Staubli VAL3: Carre10.dtx

public frame fReference = {x=1508.007, y=227.412, z=-659.53, rz=90, fatherId=world[0]}
public jointRx jPark = {j3=90, j5=90}
public jointRx jJoint = {j1=0.56611, j2=53.82368, j3=72.5366, j5=53.63971, j6=175.60048}
public mdesc mNomSpeed = {blend=off}
public mdesc mSpeed[30]
  [0] = {tmax=30, rmax=100, leave=0.1, reach=0.1, blend=cartesian}
  [1] = {tmax=30, rmax=100, leave=0.1, reach=0.1, blend=cartesian}
  [2] = {tmax=30, rmax=100, leave=0.1, reach=0.1, blend=cartesian}
  [3] = {tmax=30, rmax=100, leave=0.1, reach=0.1, blend=cartesian}
  [4] = {tmax=30, rmax=100, leave=0.1, reach=0.1, blend=cartesian}
  [5] = {tmax=30, rmax=100, leave=0.1, reach=0.1, blend=cartesian}
  [6] = {tmax=30, rmax=100, leave=0.1, reach=0.1, blend=cartesian}
  [7] = {tmax=30, rmax=100, leave=0.1, reach=0.1, blend=cartesian}
  [8] = {tmax=30, rmax=100, leave=0.1, reach=0.1, blend=cartesian}
  [9] = {tmax=30, rmax=100, leave=0.1, reach=0.1, blend=cartesian}
  [10] = {tmax=30, rmax=100, leave=0.1, reach=0.1, blend=cartesian}
  [11] = {tmax=30, rmax=100, leave=0.1, reach=0.1, blend=cartesian}
  [12] = {tmax=30, rmax=100, leave=0.1, reach=0.1, blend=cartesian}
  [13] = {tmax=30, rmax=100, leave=0.1, reach=0.1, blend=cartesian}
  [14] = {tmax=30, rmax=100, leave=0.1, reach=0.1, blend=cartesian}
  [15] = {tmax=30, rmax=100, leave=0.1, reach=0.1, blend=cartesian}
  [16] = {tmax=30, rmax=100, leave=0.1, reach=0.1, blend=cartesian}
  [17] = {tmax=30, rmax=100, leave=0.1, reach=0.1, blend=cartesian}
  [18] = {tmax=30, rmax=100, leave=0.1, reach=0.1, blend=cartesian}
  [19] = {tmax=30, rmax=100, leave=0.1, reach=0.1, blend=cartesian}
  [20] = {tmax=30, rmax=100, leave=0.1, reach=0.1, blend=cartesian}
  [21] = {tmax=30, rmax=100, leave=0.1, reach=0.1, blend=cartesian}
  [22] = {tmax=30, rmax=100, leave=0.1, reach=0.1, blend=cartesian}
  [23] = {tmax=30, rmax=100, leave=0.1, reach=0.1, blend=cartesian}
  [24] = {tmax=30, rmax=100, leave=0.1, reach=0.1, blend=cartesian}
  [25] = {tmax=30, rmax=100, leave=0.1, reach=0.1, blend=cartesian}
  [26] = {tmax=30, rmax=100, leave=0.1, reach=0.1, blend=cartesian}
  [27] = {tmax=30, rmax=100, leave=0.1, reach=0.1, blend=cartesian}
  [28] = {tmax=30, rmax=100, leave=0.1, reach=0.1, blend=cartesian}
  [29] = {tmax=30, rmax=100, leave=0.1, reach=0.1, blend=cartesian}
public num nTraj
num nTimeStop
num nTimeStart
num nMode
num nEtat
public pointRx pPoint[1630]
  [0] = {x=-211, y=-153, z=100, rx=-180, rz=85.034, shoulder=lefty, elbow=epositive, wrist=wpositive, fatherId=fReference[0]}
  [1] = {x=-211, y=-153, rx=-180, rz=85.034, shoulder=lefty, elbow=epositive, wrist=wpositive, fatherId=fReference[0]}
  [2] = {x=-211, y=-153, rx=-180, rz=85.034, shoulder=lefty, elbow=epositive, wrist=wpositive, fatherId=fReference[0]}
  [3] = {x=-210.131, y=-163.003, rx=-180, rz=75.103, shoulder=lefty, elbow=epositive, wrist=wpositive, fatherId=fReference[0]}
  [4] = {x=-207.55, y=-172.706, rx=-180, rz=65.172, shoulder=lefty, elbow=epositive, wrist=wpositive, fatherId=fReference[0]}
  [5] = {x=-203.334, y=-181.819, rx=-180, rz=55.241, shoulder=lefty, elbow=epositive, wrist=wpositive, fatherId=fReference[0]}
  [6] = {x=-197.609, y=-190.068, rx=-180, rz=45.309, shoulder=lefty, elbow=epositive, wrist=wpositive, fatherId=fReference[0]}
  [7] = {x=-190.548, y=-197.206, rx=-180, rz=35.378, shoulder=lefty, elbow=epositive, wrist=wpositive, fatherId=fReference[0]}
  [8] = {x=-182.361, y=-203.019, rx=-180, rz=25.447, shoulder=lefty, elbow=epositive, wrist=wpositive, fatherId=fReference[0]}
  [9] = {x=-173.294, y=-207.334, rx=180, rz=15.516, shoulder=lefty, elbow=epositive, wrist=wpositive, fatherId=fReference[0]}
  [10] = {x=-163.619, y=-210.02, rx=-180, rz=5.584, shoulder=lefty, elbow=epositive, wrist=wpositive, fatherId=fReference[0]}
  [11] = {x=-153.626, y=-210.997, rx=-180, rz=0.019, shoulder=lefty, elbow=epositive, wrist=wpositive, fatherId=fReference[0]}
  [12] = {x=-143.573, y=-211, rx=180, shoulder=lefty, elbow=epositive, wrist=wpositive, fatherId=fReference[0]}
  [13] = {x=-133.52, y=-211, rx=180, shoulder=lefty, elbow=epositive, wrist=wpositive, fatherId=fReference[0]}
  [14] = {x=-123.466, y=-211, rx=180, shoulder=lefty, elbow=epositive, wrist=wpositive, fatherId=fReference[0]}
  [15] = {x=-113.413, y=-211, rx=-180, shoulder=lefty, elbow=epositive, wrist=wpositive, fatherId=fReference[0]}
  [16] = {x=-103.36, y=-211, rx=180, shoulder=lefty, elbow=epositive, wrist=wpositive, fatherId=fReference[0]}
  [17] = {x=-93.306, y=-211, rx=-180, shoulder=lefty, elbow=epositive, wrist=wpositive, fatherId=fReference[0]}
  [18] = {x=-83.253, y=-211, rx=-180, shoulder=lefty, elbow=epositive, wrist=wpositive, fatherId=fReference[0]}
  [19] = {x=-73.2, y=-211, rx=-180, shoulder=lefty, elbow=epositive, wrist=wpositive, fatherId=fReference[0]}
  [20] = {x=-63.146, y=-211, rx=180, shoulder=lefty, elbow=epositive, wrist=wpositive, fatherId=fReference[0]}
  [21] = {x=-53.093, y=-211, rx=-180, shoulder=lefty, elbow=epositive, wrist=wpositive, fatherId=fReference[0]}
  [22] = {x=-43.04, y=-211, rx=180, shoulder=lefty, elbow=epositive, wrist=wpositive, fatherId=fReference[0]}
  [23] = {x=-32.986, y=-211, rx=180, shoulder=lefty, elbow=epositive, wrist=wpositive, fatherId=fReference[0]}
  [24] = {x=-22.933, y=-211, rx=-180, shoulder=lefty, elbow=epositive, wrist=wpositive, fatherId=fReference[0]}
  [25] = {x=-12.88, y=-211, rx=-180, shoulder=lefty, elbow=epositive, wrist=wpositive, fatherId=fReference[0]}
  [26] = {x=-2.826, y=-211, rx=180, shoulder=lefty, elbow=epositive, wrist=wpositive, fatherId=fReference[0]}
  [27] = {x=7.227, y=-211, rx=-180, shoulder=lefty, elbow=epositive, wrist=wpositive, fatherId=fReference[0]}
  [28] = {x=17.28, y=-211, rx=-180, shoulder=lefty, elbow=epositive, wrist=wpositive, fatherId=fReference[0]}
  [29] = {x=27.333, y=-211, rx=-180, shoulder=lefty, elbow=epositive, wrist=wpositive, fatherId=fReference[0]}
  [30] = {x=37.387, y=-211, rx=180, shoulder=lefty, elbow=epositive, wrist=wpositive, fatherId=fReference[0]}
  [31] = {x=47.44, y=-211, rx=-180, shoulder=lefty, elbow=epositive, wrist=wpositive, fatherId=fReference[0]}
  [32] = {x=57.493, y=-211, rx=180, shoulder=lefty, elbow=epositive, wrist=wpositive, fatherId=fReference[0]}
  [33] = {x=67.547, y=-211, rx=-180, shoulder=lefty, elbow=epositive, wrist=wpositive, fatherId=fReference[0]}
  [34] = {x=77.6, y=-211, rx=180, shoulder=lefty, elbow=epositive, wrist=wpositive, fatherId=fReference[0]}
  [35] = {x=87.653, y=-211, rx=-180, shoulder=lefty, elbow=epositive, wrist=wpositive, fatherId=fReference[0]}
  [36] = {x=97.707, y=-211, rx=-180, shoulder=lefty, elbow=epositive, wrist=wpositive, fatherId=fReference[0]}
  [37] = {x=107.76, y=-211, rx=180, shoulder=lefty, elbow=epositive, wrist=wpositive, fatherId=fReference[0]}
  [38] = {x=117.813, y=-211, rx=180, shoulder=lefty, elbow=epositive, wrist=wpositive, fatherId=fReference[0]}
  [39] = {x=127.867, y=-211, rx=-180, shoulder=lefty, elbow=epositive, wrist=wpositive, fatherId=fReference[0]}
  [40] = {x=137.92, y=-211, rx=-180, shoulder=lefty, elbow=epositive, wrist=wpositive, fatherId=fReference[0]}
  [41] = {x=147.973, y=-211, rx=-180, rz=-1.241, shoulder=lefty, elbow=epositive, wrist=wpositive, fatherId=fReference[0]}
  [42] = {x=158.02, y=-210.782, rx=-180, rz=-9.931, shoulder=lefty, elbow=epositive, wrist=wpositive, fatherId=fReference[0]}
  [43] = {x=167.911, y=-209.051, rx=-180, rz=-19.863, shoulder=lefty, elbow=epositive, wrist=wpositive, fatherId=fReference[0]}
  [44] = {x=177.354, y=-205.639, rx=-180, rz=-29.794, shoulder=lefty, elbow=epositive, wrist=wpositive, fatherId=fReference[0]}
  [45] = {x=186.068, y=-200.65, rx=180, rz=-39.725, shoulder=lefty, elbow=epositive, wrist=wpositive, fatherId=fReference[0]}
  [46] = {x=193.79, y=-194.233, rx=180, rz=-49.656, shoulder=lefty, elbow=epositive, wrist=wpositive, fatherId=fReference[0]}
  [47] = {x=200.29, y=-186.58, rx=180, rz=-59.588, shoulder=lefty, elbow=epositive, wrist=wpositive, fatherId=fReference[0]}
  [48] = {x=205.373, y=-177.921, rx=180, rz=-69.519, shoulder=lefty, elbow=epositive, wrist=wpositive, fatherId=fReference[0]}
  [49] = {x=208.886, y=-168.515, rx=180, rz=-79.45, shoulder=lefty, elbow=epositive, wrist=wpositive, fatherId=fReference[0]}
  [50] = {x=210.725, y=-158.644, rx=180, rz=-88.43, shoulder=lefty, elbow=epositive, wrist=wpositive, fatherId=fReference[0]}
  [51] = {x=211, y=-148.6, rx=180, rz=-90, shoulder=lefty, elbow=epositive, wrist=wpositive, fatherId=fReference[0]}
  [52] = {x=211, y=-138.546, rx=180, rz=-90, shoulder=lefty, elbow=epositive, wrist=wpositive, fatherId=fReference[0]}
  [53] = {x=211, y=-128.493, rx=180, rz=-90, shoulder=lefty, elbow=epositive, wrist=wpositive, fatherId=fReference[0]}
  [54] = {x=211, y=-118.44, rx=180, rz=-90, shoulder=lefty, elbow=epositive, wrist=wpositive, fatherId=fReference[0]}
  [55] = {x=211, y=-108.386, rx=180, rz=-90, shoulder=lefty, elbow=epositive, wrist=wpositive, fatherId=fReference[0]}
  [56] = {x=211, y=-98.333, rx=180, rz=-90, shoulder=lefty, elbow=epositive, wrist=wpositive, fatherId=fReference[0]}
  [57] = {x=211, y=-88.28, rx=180, rz=-90, shoulder=lefty, elbow=epositive, wrist=wpositive, fatherId=fReference[0]}
  [58] = {x=211, y=-78.226, rx=180, rz=-90, shoulder=lefty, elbow=epositive, wrist=wpositive, fatherId=fReference[0]}
  [59] = {x=211, y=-68.173, rx=180, rz=-90, shoulder=lefty, elbow=epositive, wrist=wpositive, fatherId=fReference[0]}
  [60] = {x=211, y=-58.12, rx=180, rz=-90, shoulder=lefty, elbow=epositive, wrist=wpositive, fatherId=fReference[0]}
  [61] = {x=211, y=-48.066, rx=180, rz=-90, shoulder=lefty, elbow=epositive, wrist=wpositive, fatherId=fReference[0]}
  [62] = {x=211, y=-38.013, rx=180, rz=-90, shoulder=lefty, elbow=epositive, wrist=wpositive, fatherId=fReference[0]}
  [63] = {x=211, y=-27.96, rx=180, rz=-90, shoulder=lefty, elbow=epositive, wrist=wpositive, fatherId=fReference[0]}
  [64] = {x=211, y=-17.906, rx=180, rz=-90, shoulder=lefty, elbow=epositive, wrist=wpositive, fatherId=fReference[0]}
  [65] = {x=211, y=-7.853, rx=180, rz=-90, shoulder=lefty, elbow=epositive, wrist=wpositive, fatherId=fReference[0]}
  [66] = {x=211, y=2.2, rx=180, rz=-90, shoulder=lefty, elbow=epositive, wrist=wpositive, fatherId=fReference[0]}
  [67] = {x=211, y=12.254, rx=180, rz=-90, shoulder=lefty, elbow=epositive, wrist=wpositive, fatherId=fReference[0]}
  [68] = {x=211, y=22.307, rx=180, rz=-90, shoulder=lefty, elbow=epositive, wrist=wpositive, fatherId=fReference[0]}
  [69] = {x=211, y=32.36, rx=180, rz=-90, shoulder=lefty, elbow=epositive, wrist=wpositive, fatherId=fReference[0]}
  [70] = {x=211, y=42.413, rx=180, rz=-90, shoulder=lefty, elbow=epositive, wrist=wpositive, fatherId=fReference[0]}
  [71] = {x=211, y=52.467, rx=180, rz=-90, shoulder=lefty, elbow=epositive, wrist=wpositive, fatherId=fReference[0]}
  [72] = {x=211, y=62.52, rx=180, rz=-90, shoulder=lefty, elbow=epositive, wrist=wpositive, fatherId=fReference[0]}
  [73] = {x=211, y=72.573, rx=180, rz=-90, shoulder=lefty, elbow=epositive, wrist=wpositive, fatherId=fReference[0]}
  [74] = {x=211, y=82.627, rx=180, rz=-90, shoulder=lefty, elbow=epositive, wrist=wpositive, fatherId=fReference[0]}
  [75] = {x=211, y=92.68, rx=180, rz=-90, shoulder=lefty, elbow=epositive, wrist=wpositive, fatherId=fReference[0]}
  [76] = {x=211, y=102.733, rx=180, rz=-90, shoulder=lefty, elbow=epositive, wrist=wpositive, fatherId=fReference[0]}
  [77] = {x=211, y=112.787, rx=180, rz=-90, shoulder=lefty, elbow=epositive, wrist=wpositive, fatherId=fReference[0]}
  [78] = {x=211, y=122.84, rx=180, rz=-90, shoulder=lefty, elbow=epositive, wrist=wpositive, fatherId=fReference[0]}
  [79] = {x=211, y=132.893, rx=180, rz=-90, shoulder=lefty, elbow=epositive, wrist=wpositive, fatherId=fReference[0]}
  [80] = {x=211, y=142.947, rx=180, rz=-90, shoulder=lefty, elbow=epositive, wrist=wpositive, fatherId=fReference[0]}
  [81] = {x=211, y=153, rx=-180, rz=-94.966, shoulder=lefty, elbow=epositive, wrist=wpositive, fatherId=fReference[0]}
  [82] = {x=210.131, y=163.003, rx=-180, rz=-104.897, shoulder=lefty, elbow=epositive, wrist=wpositive, fatherId=fReference[0]}
  [83] = {x=207.55, y=172.706, rx=-180, rz=-114.828, shoulder=lefty, elbow=epositive, wrist=wpositive, fatherId=fReference[0]}
  [84] = {x=203.334, y=181.819, rx=-180, rz=-124.759, shoulder=lefty, elbow=epositive, wrist=wpositive, fatherId=fReference[0]}
  [85] = {x=197.609, y=190.068, rx=-180, rz=-134.691, shoulder=lefty, elbow=epositive, wrist=wpositive, fatherId=fReference[0]}
  [86] = {x=190.548, y=197.206, rx=180, rz=-144.622, shoulder=lefty, elbow=epositive, wrist=wpositive, fatherId=fReference[0]}
  [87] = {x=182.361, y=203.019, rx=-180, rz=-154.553, shoulder=lefty, elbow=epositive, wrist=wpositive, fatherId=fReference[0]}
  [88] = {x=173.294, y=207.334, rx=-180, rz=-164.484, shoulder=lefty, elbow=epositive, wrist=wpositive, fatherId=fReference[0]}
  [89] = {x=163.619, y=210.02, rx=-180, rz=-174.416, shoulder=lefty, elbow=epositive, wrist=wpositive, fatherId=fReference[0]}
  [90] = {x=153.626, y=210.997, rx=-180, rz=-179.981, shoulder=lefty, elbow=epositive, wrist=wpositive, fatherId=fReference[0]}
  [91] = {x=143.573, y=211, rx=180, rz=-180, shoulder=lefty, elbow=epositive, wrist=wpositive, fatherId=fReference[0]}
  [92] = {x=133.52, y=211, rx=-180, rz=180, shoulder=lefty, elbow=epositive, wrist=wpositive, fatherId=fReference[0]}
  [93] = {x=123.466, y=211, rx=-180, rz=180, shoulder=lefty, elbow=epositive, wrist=wpositive, fatherId=fReference[0]}
  [94] = {x=113.413, y=211, rx=180, rz=-180, shoulder=lefty, elbow=epositive, wrist=wpositive, fatherId=fReference[0]}
  [95] = {x=103.36, y=211, rx=180, rz=180, shoulder=lefty, elbow=epositive, wrist=wpositive, fatherId=fReference[0]}
  [96] = {x=93.306, y=211, rx=-180, rz=180, shoulder=lefty, elbow=epositive, wrist=wpositive, fatherId=fReference[0]}
  [97] = {x=83.253, y=211, rx=-180, rz=-180, shoulder=lefty, elbow=epositive, wrist=wpositive, fatherId=fReference[0]}
  [98] = {x=73.2, y=211, rx=180, rz=180, shoulder=lefty, elbow=epositive, wrist=wpositive, fatherId=fReference[0]}
  [99] = {x=63.146, y=211, rx=-180, rz=180, shoulder=lefty, elbow=epositive, wrist=wpositive, fatherId=fReference[0]}
  [100] = {x=53.093, y=211, rx=-180, rz=180, shoulder=lefty, elbow=epositive, wrist=wpositive, fatherId=fReference[0]}
  [101] = {x=43.04, y=211, rx=-180, rz=180, shoulder=lefty, elbow=epositive, wrist=wpositive, fatherId=fReference[0]}
  [102] = {x=32.986, y=211, rx=-180, rz=180, shoulder=lefty, elbow=epositive, wrist=wpositive, fatherId=fReference[0]}
  [103] = {x=22.933, y=211, rx=-180, rz=180, shoulder=lefty, elbow=epositive, wrist=wpositive, fatherId=fReference[0]}
  [104] = {x=12.88, y=211, rx=180, rz=180, shoulder=lefty, elbow=epositive, wrist=wpositive, fatherId=fReference[0]}
  [105] = {x=2.826, y=211, rx=180, rz=180, shoulder=lefty, elbow=epositive, wrist=wpositive, fatherId=fReference[0]}
  [106] = {x=-7.227, y=211, rx=-180, rz=180, shoulder=lefty, elbow=epositive, wrist=wpositive, fatherId=fReference[0]}
  [107] = {x=-17.28, y=211, rx=180, rz=180, shoulder=lefty, elbow=epositive, wrist=wpositive, fatherId=fReference[0]}
  [108] = {x=-27.333, y=211, rx=180, rz=180, shoulder=lefty, elbow=epositive, wrist=wpositive, fatherId=fReference[0]}
  [109] = {x=-37.387, y=211, rx=-180, rz=180, shoulder=lefty, elbow=epositive, wrist=wpositive, fatherId=fReference[0]}
  [110] = {x=-47.44, y=211, rx=180, rz=180, shoulder=lefty, elbow=epositive, wrist=wpositive, fatherId=fReference[0]}
  [111] = {x=-57.493, y=211, rx=-180, rz=180, shoulder=lefty, elbow=epositive, wrist=wpositive, fatherId=fReference[0]}
  [112] = {x=-67.547, y=211, rx=180, rz=180, shoulder=lefty, elbow=epositive, wrist=wpositive, fatherId=fReference[0]}
  [113] = {x=-77.6, y=211, rx=-180, rz=180, shoulder=lefty, elbow=epositive, wrist=wpositive, fatherId=fReference[0]}
  [114] = {x=-87.653, y=211, rx=180, rz=180, shoulder=lefty, elbow=epositive, wrist=wpositive, fatherId=fReference[0]}
  [115] = {x=-97.707, y=211, rx=180, rz=180, shoulder=lefty, elbow=epositive, wrist=wpositive, fatherId=fReference[0]}
  [116] = {x=-107.76, y=211, rx=180, rz=180, shoulder=lefty, elbow=epositive, wrist=wpositive, fatherId=fReference[0]}
  [117] = {x=-117.813, y=211, rx=-180, rz=180, shoulder=lefty, elbow=epositive, wrist=wpositive, fatherId=fReference[0]}
  [118] = {x=-127.867, y=211, rx=-180, rz=180, shoulder=lefty, elbow=epositive, wrist=wpositive, fatherId=fReference[0]}
  [119] = {x=-137.92, y=211, rx=180, rz=180, shoulder=lefty, elbow=epositive, wrist=wpositive, fatherId=fReference[0]}
  [120] = {x=-147.973, y=211, rx=180, rz=178.759, shoulder=lefty, elbow=epositive, wrist=wpositive, fatherId=fReference[0]}
  [121] = {x=-158.02, y=210.782, rx=180, rz=170.069, shoulder=lefty, elbow=epositive, wrist=wpositive, fatherId=fReference[0]}
  [122] = {x=-167.911, y=209.051, rx=180, rz=160.137, shoulder=lefty, elbow=epositive, wrist=wpositive, fatherId=fReference[0]}
  [123] = {x=-177.354, y=205.639, rx=180, rz=150.206, shoulder=lefty, elbow=epositive, wrist=wpositive, fatherId=fReference[0]}
  [124] = {x=-186.068, y=200.65, rx=180, rz=140.275, shoulder=lefty, elbow=epositive, wrist=wpositive, fatherId=fReference[0]}
  [125] = {x=-193.79, y=194.233, rx=-180, rz=130.344, shoulder=lefty, elbow=epositive, wrist=wpositive, fatherId=fReference[0]}
  [126] = {x=-200.29, y=186.58, rx=180, rz=120.412, shoulder=lefty, elbow=epositive, wrist=wpositive, fatherId=fReference[0]}
  [127] = {x=-205.373, y=177.921, rx=180, rz=110.481, shoulder=lefty, elbow=epositive, wrist=wpositive, fatherId=fReference[0]}
  [128] = {x=-208.886, y=168.515, rx=180, rz=100.55, shoulder=lefty, elbow=epositive, wrist=wpositive, fatherId=fReference[0]}
  [129] = {x=-210.725, y=158.644, rx=180, rz=91.57, shoulder=lefty, elbow=epositive, wrist=wpositive, fatherId=fReference[0]}
  [130] = {x=-211, y=148.6, rx=-180, rz=90, shoulder=lefty, elbow=epositive, wrist=wpositive, fatherId=fReference[0]}
  [131] = {x=-211, y=138.546, rx=-180, rz=90, shoulder=lefty, elbow=epositive, wrist=wpositive, fatherId=fReference[0]}
  [132] = {x=-211, y=128.493, rx=-180, rz=90, shoulder=lefty, elbow=epositive, wrist=wpositive, fatherId=fReference[0]}
  [133] = {x=-211, y=118.44, rx=-180, rz=90, shoulder=lefty, elbow=epositive, wrist=wpositive, fatherId=fReference[0]}
  [134] = {x=-211, y=108.386, rx=-180, rz=90, shoulder=lefty, elbow=epositive, wrist=wpositive, fatherId=fReference[0]}
  [135] = {x=-211, y=98.333, rx=-180, rz=90, shoulder=lefty, elbow=epositive, wrist=wpositive, fatherId=fReference[0]}
  [136] = {x=-211, y=88.28, rx=-180, rz=90, shoulder=lefty, elbow=epositive, wrist=wpositive, fatherId=fReference[0]}
  [137] = {x=-211, y=78.226, rx=-180, rz=90, shoulder=lefty, elbow=epositive, wrist=wpositive, fatherId=fReference[0]}
  [138] = {x=-211, y=68.173, rx=-180, rz=90, shoulder=lefty, elbow=epositive, wrist=wpositive, fatherId=fReference[0]}
  [139] = {x=-211, y=58.12, rx=-180, rz=90, shoulder=lefty, elbow=epositive, wrist=wpositive, fatherId=fReference[0]}
  [140] = {x=-211, y=48.066, rx=-180, rz=90, shoulder=lefty, elbow=epositive, wrist=wpositive, fatherId=fReference[0]}
  [141] = {x=-211, y=38.013, rx=-180, rz=90, shoulder=lefty, elbow=epositive, wrist=wpositive, fatherId=fReference[0]}
  [142] = {x=-211, y=27.96, rx=-180, rz=90, shoulder=lefty, elbow=epositive, wrist=wpositive, fatherId=fReference[0]}
  [143] = {x=-211, y=17.906, rx=-180, rz=90, shoulder=lefty, elbow=epositive, wrist=wpositive, fatherId=fReference[0]}
  [144] = {x=-211, y=7.853, rx=-180, rz=90, shoulder=lefty, elbow=epositive, wrist=wpositive, fatherId=fReference[0]}
  [145] = {x=-211, y=-2.2, rx=-180, rz=90, shoulder=lefty, elbow=epositive, wrist=wpositive, fatherId=fReference[0]}
  [146] = {x=-211, y=-12.254, rx=-180, rz=90, shoulder=lefty, elbow=epositive, wrist=wpositive, fatherId=fReference[0]}
  [147] = {x=-211, y=-22.307, rx=-180, rz=90, shoulder=lefty, elbow=epositive, wrist=wpositive, fatherId=fReference[0]}
  [148] = {x=-211, y=-32.36, rx=-180, rz=90, shoulder=lefty, elbow=epositive, wrist=wpositive, fatherId=fReference[0]}
  [149] = {x=-211, y=-42.413, rx=-180, rz=90, shoulder=lefty, elbow=epositive, wrist=wpositive, fatherId=fReference[0]}
  [150] = {x=-211, y=-52.467, rx=-180, rz=90, shoulder=lefty, elbow=epositive, wrist=wpositive, fatherId=fReference[0]}
  [151] = {x=-211, y=-62.52, rx=-180, rz=90, shoulder=lefty, elbow=epositive, wrist=wpositive, fatherId=fReference[0]}
  [152] = {x=-211, y=-72.573, rx=-180, rz=90, shoulder=lefty, elbow=epositive, wrist=wpositive, fatherId=fReference[0]}
  [153] = {x=-211, y=-82.627, rx=-180, rz=90, shoulder=lefty, elbow=epositive, wrist=wpositive, fatherId=fReference[0]}
  [154] = {x=-211, y=-92.68, rx=-180, rz=90, shoulder=lefty, elbow=epositive, wrist=wpositive, fatherId=fReference[0]}
  [155] = {x=-211, y=-102.733, rx=-180, rz=90, shoulder=lefty, elbow=epositive, wrist=wpositive, fatherId=fReference[0]}
  [156] = {x=-211, y=-112.787, rx=-180, rz=90, shoulder=lefty, elbow=epositive, wrist=wpositive, fatherId=fReference[0]}
  [157] = {x=-211, y=-122.84, rx=-180, rz=90, shoulder=lefty, elbow=epositive, wrist=wpositive, fatherId=fReference[0]}
  [158] = {x=-211, y=-132.893, rx=-180, rz=90, shoulder=lefty, elbow=epositive, wrist=wpositive, fatherId=fReference[0]}
  [159] = {x=-211, y=-142.947, rx=-180, rz=90, shoulder=lefty, elbow=epositive, wrist=wpositive, fatherId=fReference[0]}
  [160] = {x=-211, y=-153, rx=-180, rz=90, shoulder=lefty, elbow=epositive, wrist=wpositive, fatherId=fReference[0]}
  [161] = {x=-211, y=-153, rx=-180, rz=90, shoulder=lefty, elbow=epositive, wrist=wpositive, fatherId=fReference[0]}
  [162] = {x=-211, y=-153, z=100, rx=-180, rz=90, shoulder=lefty, elbow=epositive, wrist=wpositive, fatherId=fReference[0]}
  [163] = {x=-211, y=-153, z=122, rx=-180, rz=90, shoulder=lefty, elbow=epositive, wrist=wpositive, fatherId=fReference[0]}
  [164] = {x=-211, y=-153, z=22, rx=-180, rz=90, shoulder=lefty, elbow=epositive, wrist=wpositive, fatherId=fReference[0]}
  [165] = {x=-211, y=-153, z=22, rx=-180, rz=90, shoulder=lefty, elbow=epositive, wrist=wpositive, fatherId=fReference[0]}
  [166] = {x=-211, y=-142.947, z=22, rx=-180, rz=90, shoulder=lefty, elbow=epositive, wrist=wpositive, fatherId=fReference[0]}
  [167] = {x=-211, y=-132.893, z=22, rx=-180, rz=90, shoulder=lefty, elbow=epositive, wrist=wpositive, fatherId=fReference[0]}
  [168] = {x=-211, y=-122.84, z=22, rx=-180, rz=90, shoulder=lefty, elbow=epositive, wrist=wpositive, fatherId=fReference[0]}
  [169] = {x=-211, y=-112.787, z=22, rx=-180, rz=90, shoulder=lefty, elbow=epositive, wrist=wpositive, fatherId=fReference[0]}
  [170] = {x=-211, y=-102.733, z=22, rx=-180, rz=90, shoulder=lefty, elbow=epositive, wrist=wpositive, fatherId=fReference[0]}
  [171] = {x=-211, y=-92.68, z=22, rx=-180, rz=90, shoulder=lefty, elbow=epositive, wrist=wpositive, fatherId=fReference[0]}
  [172] = {x=-211, y=-82.627, z=22, rx=-180, rz=90, shoulder=lefty, elbow=epositive, wrist=wpositive, fatherId=fReference[0]}
  [173] = {x=-211, y=-72.573, z=22, rx=-180, rz=90, shoulder=lefty, elbow=epositive, wrist=wpositive, fatherId=fReference[0]}
  [174] = {x=-211, y=-62.52, z=22, rx=-180, rz=90, shoulder=lefty, elbow=epositive, wrist=wpositive, fatherId=fReference[0]}
  [175] = {x=-211, y=-52.467, z=22, rx=-180, rz=90, shoulder=lefty, elbow=epositive, wrist=wpositive, fatherId=fReference[0]}
  [176] = {x=-211, y=-42.413, z=22, rx=-180, rz=90, shoulder=lefty, elbow=epositive, wrist=wpositive, fatherId=fReference[0]}
  [177] = {x=-211, y=-32.36, z=22, rx=-180, rz=90, shoulder=lefty, elbow=epositive, wrist=wpositive, fatherId=fReference[0]}
  [178] = {x=-211, y=-22.307, z=22, rx=-180, rz=90, shoulder=lefty, elbow=epositive, wrist=wpositive, fatherId=fReference[0]}
  [179] = {x=-211, y=-12.254, z=22, rx=-180, rz=90, shoulder=lefty, elbow=epositive, wrist=wpositive, fatherId=fReference[0]}
  [180] = {x=-211, y=-2.2, z=22, rx=-180, rz=90, shoulder=lefty, elbow=epositive, wrist=wpositive, fatherId=fReference[0]}
  [181] = {x=-211, y=7.853, z=22, rx=-180, rz=90, shoulder=lefty, elbow=epositive, wrist=wpositive, fatherId=fReference[0]}
  [182] = {x=-211, y=17.906, z=22, rx=-180, rz=90, shoulder=lefty, elbow=epositive, wrist=wpositive, fatherId=fReference[0]}
  [183] = {x=-211, y=27.96, z=22, rx=-180, rz=90, shoulder=lefty, elbow=epositive, wrist=wpositive, fatherId=fReference[0]}
  [184] = {x=-211, y=38.013, z=22, rx=-180, rz=90, shoulder=lefty, elbow=epositive, wrist=wpositive, fatherId=fReference[0]}
  [185] = {x=-211, y=48.066, z=22, rx=-180, rz=90, shoulder=lefty, elbow=epositive, wrist=wpositive, fatherId=fReference[0]}
  [186] = {x=-211, y=58.12, z=22, rx=-180, rz=90, shoulder=lefty, elbow=epositive, wrist=wpositive, fatherId=fReference[0]}
  [187] = {x=-211, y=68.173, z=22, rx=-180, rz=90, shoulder=lefty, elbow=epositive, wrist=wpositive, fatherId=fReference[0]}
  [188] = {x=-211, y=78.226, z=22, rx=-180, rz=90, shoulder=lefty, elbow=epositive, wrist=wpositive, fatherId=fReference[0]}
  [189] = {x=-211, y=88.28, z=22, rx=-180, rz=90, shoulder=lefty, elbow=epositive, wrist=wpositive, fatherId=fReference[0]}
  [190] = {x=-211, y=98.333, z=22, rx=-180, rz=90, shoulder=lefty, elbow=epositive, wrist=wpositive, fatherId=fReference[0]}
  [191] = {x=-211, y=108.386, z=22, rx=-180, rz=90, shoulder=lefty, elbow=epositive, wrist=wpositive, fatherId=fReference[0]}
  [192] = {x=-211, y=118.44, z=22, rx=-180, rz=90, shoulder=lefty, elbow=epositive, wrist=wpositive, fatherId=fReference[0]}
  [193] = {x=-211, y=128.493, z=22, rx=-180, rz=90, shoulder=lefty, elbow=epositive, wrist=wpositive, fatherId=fReference[0]}
  [194] = {x=-211, y=138.546, z=22, rx=-180, rz=90, shoulder=lefty, elbow=epositive, wrist=wpositive, fatherId=fReference[0]}
  [195] = {x=-211, y=148.6, z=22, rx=180, rz=91.57, shoulder=lefty, elbow=epositive, wrist=wpositive, fatherId=fReference[0]}
  [196] = {x=-210.725, y=158.644, z=22, rx=180, rz=100.55, shoulder=lefty, elbow=epositive, wrist=wpositive, fatherId=fReference[0]}
  [197] = {x=-208.886, y=168.515, z=22, rx=180, rz=110.481, shoulder=lefty, elbow=epositive, wrist=wpositive, fatherId=fReference[0]}
  [198] = {x=-205.373, y=177.921, z=22, rx=180, rz=120.412, shoulder=lefty, elbow=epositive, wrist=wpositive, fatherId=fReference[0]}
  [199] = {x=-200.29, y=186.58, z=22, rx=-180, rz=130.344, shoulder=lefty, elbow=epositive, wrist=wpositive, fatherId=fReference[0]}
  [200] = {x=-193.79, y=194.233, z=22, rx=-180, rz=140.275, shoulder=lefty, elbow=epositive, wrist=wpositive, fatherId=fReference[0]}
  [201] = {x=-186.068, y=200.65, z=22, rx=180, rz=150.206, shoulder=lefty, elbow=epositive, wrist=wpositive, fatherId=fReference[0]}
  [202] = {x=-177.354, y=205.639, z=22, rx=180, rz=160.137, shoulder=lefty, elbow=epositive, wrist=wpositive, fatherId=fReference[0]}
  [203] = {x=-167.911, y=209.051, z=22, rx=180, rz=170.069, shoulder=lefty, elbow=epositive, wrist=wpositive, fatherId=fReference[0]}
  [204] = {x=-158.02, y=210.782, z=22, rx=180, rz=178.759, shoulder=lefty, elbow=epositive, wrist=wpositive, fatherId=fReference[0]}
  [205] = {x=-147.973, y=211, z=22, rx=-180, rz=180, shoulder=lefty, elbow=epositive, wrist=wpositive, fatherId=fReference[0]}
  [206] = {x=-137.92, y=211, z=22, rx=-180, rz=180, shoulder=lefty, elbow=epositive, wrist=wpositive, fatherId=fReference[0]}
  [207] = {x=-127.867, y=211, z=22, rx=-180, rz=180, shoulder=lefty, elbow=epositive, wrist=wpositive, fatherId=fReference[0]}
  [208] = {x=-117.813, y=211, z=22, rx=180, rz=180, shoulder=lefty, elbow=epositive, wrist=wpositive, fatherId=fReference[0]}
  [209] = {x=-107.76, y=211, z=22, rx=180, rz=180, shoulder=lefty, elbow=epositive, wrist=wpositive, fatherId=fReference[0]}
  [210] = {x=-97.707, y=211, z=22, rx=-180, rz=180, shoulder=lefty, elbow=epositive, wrist=wpositive, fatherId=fReference[0]}
  [211] = {x=-87.653, y=211, z=22, rx=-180, rz=180, shoulder=lefty, elbow=epositive, wrist=wpositive, fatherId=fReference[0]}
  [212] = {x=-77.6, y=211, z=22, rx=-180, rz=180, shoulder=lefty, elbow=epositive, wrist=wpositive, fatherId=fReference[0]}
  [213] = {x=-67.547, y=211, z=22, rx=-180, rz=180, shoulder=lefty, elbow=epositive, wrist=wpositive, fatherId=fReference[0]}
  [214] = {x=-57.493, y=211, z=22, rx=180, rz=180, shoulder=lefty, elbow=epositive, wrist=wpositive, fatherId=fReference[0]}
  [215] = {x=-47.44, y=211, z=22, rx=180, rz=180, shoulder=lefty, elbow=epositive, wrist=wpositive, fatherId=fReference[0]}
  [216] = {x=-37.387, y=211, z=22, rx=-180, rz=180, shoulder=lefty, elbow=epositive, wrist=wpositive, fatherId=fReference[0]}
  [217] = {x=-27.333, y=211, z=22, rx=-180, rz=180, shoulder=lefty, elbow=epositive, wrist=wpositive, fatherId=fReference[0]}
  [218] = {x=-17.28, y=211, z=22, rx=180, rz=180, shoulder=lefty, elbow=epositive, wrist=wpositive, fatherId=fReference[0]}
  [219] = {x=-7.227, y=211, z=22, rx=-180, rz=180, shoulder=lefty, elbow=epositive, wrist=wpositive, fatherId=fReference[0]}
  [220] = {x=2.826, y=211, z=22, rx=-180, rz=180, shoulder=lefty, elbow=epositive, wrist=wpositive, fatherId=fReference[0]}
  [221] = {x=12.88, y=211, z=22, rx=-180, rz=180, shoulder=lefty, elbow=epositive, wrist=wpositive, fatherId=fReference[0]}
  [222] = {x=22.933, y=211, z=22, rx=180, rz=180, shoulder=lefty, elbow=epositive, wrist=wpositive, fatherId=fReference[0]}
  [223] = {x=32.986, y=211, z=22, rx=180, rz=180, shoulder=lefty, elbow=epositive, wrist=wpositive, fatherId=fReference[0]}
  [224] = {x=43.04, y=211, z=22, rx=-180, rz=180, shoulder=lefty, elbow=epositive, wrist=wpositive, fatherId=fReference[0]}
  [225] = {x=53.093, y=211, z=22, rx=-180, rz=180, shoulder=lefty, elbow=epositive, wrist=wpositive, fatherId=fReference[0]}
  [226] = {x=63.146, y=211, z=22, rx=-180, rz=180, shoulder=lefty, elbow=epositive, wrist=wpositive, fatherId=fReference[0]}
  [227] = {x=73.2, y=211, z=22, rx=180, rz=180, shoulder=lefty, elbow=epositive, wrist=wpositive, fatherId=fReference[0]}
  [228] = {x=83.253, y=211, z=22, rx=180, rz=-180, shoulder=lefty, elbow=epositive, wrist=wpositive, fatherId=fReference[0]}
  [229] = {x=93.306, y=211, z=22, rx=-180, rz=180, shoulder=lefty, elbow=epositive, wrist=wpositive, fatherId=fReference[0]}
  [230] = {x=103.36, y=211, z=22, rx=180, rz=180, shoulder=lefty, elbow=epositive, wrist=wpositive, fatherId=fReference[0]}
  [231] = {x=113.413, y=211, z=22, rx=180, rz=-180, shoulder=lefty, elbow=epositive, wrist=wpositive, fatherId=fReference[0]}
  [232] = {x=123.466, y=211, z=22, rx=180, rz=180, shoulder=lefty, elbow=epositive, wrist=wpositive, fatherId=fReference[0]}
  [233] = {x=133.52, y=211, z=22, rx=-180, rz=180, shoulder=lefty, elbow=epositive, wrist=wpositive, fatherId=fReference[0]}
  [234] = {x=143.573, y=211, z=22, rx=-180, rz=-179.981, shoulder=lefty, elbow=epositive, wrist=wpositive, fatherId=fReference[0]}
  [235] = {x=153.626, y=210.997, z=22, rx=-180, rz=-174.416, shoulder=lefty, elbow=epositive, wrist=wpositive, fatherId=fReference[0]}
  [236] = {x=163.619, y=210.02, z=22, rx=180, rz=-164.484, shoulder=lefty, elbow=epositive, wrist=wpositive, fatherId=fReference[0]}
  [237] = {x=173.294, y=207.334, z=22, rx=-180, rz=-154.553, shoulder=lefty, elbow=epositive, wrist=wpositive, fatherId=fReference[0]}
  [238] = {x=182.361, y=203.019, z=22, rx=-180, rz=-144.622, shoulder=lefty, elbow=epositive, wrist=wpositive, fatherId=fReference[0]}
  [239] = {x=190.548, y=197.206, z=22, rx=-180, rz=-134.691, shoulder=lefty, elbow=epositive, wrist=wpositive, fatherId=fReference[0]}
  [240] = {x=197.609, y=190.068, z=22, rx=-180, rz=-124.759, shoulder=lefty, elbow=epositive, wrist=wpositive, fatherId=fReference[0]}
  [241] = {x=203.334, y=181.819, z=22, rx=-180, rz=-114.828, shoulder=lefty, elbow=epositive, wrist=wpositive, fatherId=fReference[0]}
  [242] = {x=207.55, y=172.706, z=22, rx=-180, rz=-104.897, shoulder=lefty, elbow=epositive, wrist=wpositive, fatherId=fReference[0]}
  [243] = {x=210.131, y=163.003, z=22, rx=-180, rz=-94.966, shoulder=lefty, elbow=epositive, wrist=wpositive, fatherId=fReference[0]}
  [244] = {x=211, y=153, z=22, rx=180, rz=-90, shoulder=lefty, elbow=epositive, wrist=wpositive, fatherId=fReference[0]}
  [245] = {x=211, y=142.947, z=22, rx=180, rz=-90, shoulder=lefty, elbow=epositive, wrist=wpositive, fatherId=fReference[0]}
  [246] = {x=211, y=132.893, z=22, rx=180, rz=-90, shoulder=lefty, elbow=epositive, wrist=wpositive, fatherId=fReference[0]}
  [247] = {x=211, y=122.84, z=22, rx=-180, rz=-90, shoulder=lefty, elbow=epositive, wrist=wpositive, fatherId=fReference[0]}
  [248] = {x=211, y=112.787, z=22, rx=180, rz=-90, shoulder=lefty, elbow=epositive, wrist=wpositive, fatherId=fReference[0]}
  [249] = {x=211, y=102.733, z=22, rx=180, rz=-90, shoulder=lefty, elbow=epositive, wrist=wpositive, fatherId=fReference[0]}
  [250] = {x=211, y=92.68, z=22, rx=180, rz=-90, shoulder=lefty, elbow=epositive, wrist=wpositive, fatherId=fReference[0]}
  [251] = {x=211, y=82.627, z=22, rx=180, rz=-90, shoulder=lefty, elbow=epositive, wrist=wpositive, fatherId=fReference[0]}
  [252] = {x=211, y=72.573, z=22, rx=180, rz=-90, shoulder=lefty, elbow=epositive, wrist=wpositive, fatherId=fReference[0]}
  [253] = {x=211, y=62.52, z=22, rx=180, rz=-90, shoulder=lefty, elbow=epositive, wrist=wpositive, fatherId=fReference[0]}
  [254] = {x=211, y=52.467, z=22, rx=180, rz=-90, shoulder=lefty, elbow=epositive, wrist=wpositive, fatherId=fReference[0]}
  [255] = {x=211, y=42.413, z=22, rx=180, rz=-90, shoulder=lefty, elbow=epositive, wrist=wpositive, fatherId=fReference[0]}
  [256] = {x=211, y=32.36, z=22, rx=180, rz=-90, shoulder=lefty, elbow=epositive, wrist=wpositive, fatherId=fReference[0]}
  [257] = {x=211, y=22.307, z=22, rx=180, rz=-90, shoulder=lefty, elbow=epositive, wrist=wpositive, fatherId=fReference[0]}
  [258] = {x=211, y=12.254, z=22, rx=180, rz=-90, shoulder=lefty, elbow=epositive, wrist=wpositive, fatherId=fReference[0]}
  [259] = {x=211, y=2.2, z=22, rx=180, rz=-90, shoulder=lefty, elbow=epositive, wrist=wpositive, fatherId=fReference[0]}
  [260] = {x=211, y=-7.853, z=22, rx=180, rz=-90, shoulder=lefty, elbow=epositive, wrist=wpositive, fatherId=fReference[0]}
  [261] = {x=211, y=-17.906, z=22, rx=180, rz=-90, shoulder=lefty, elbow=epositive, wrist=wpositive, fatherId=fReference[0]}
  [262] = {x=211, y=-27.96, z=22, rx=180, rz=-90, shoulder=lefty, elbow=epositive, wrist=wpositive, fatherId=fReference[0]}
  [263] = {x=211, y=-38.013, z=22, rx=180, rz=-90, shoulder=lefty, elbow=epositive, wrist=wpositive, fatherId=fReference[0]}
  [264] = {x=211, y=-48.066, z=22, rx=180, rz=-90, shoulder=lefty, elbow=epositive, wrist=wpositive, fatherId=fReference[0]}
  [265] = {x=211, y=-58.12, z=22, rx=180, rz=-90, shoulder=lefty, elbow=epositive, wrist=wpositive, fatherId=fReference[0]}
  [266] = {x=211, y=-68.173, z=22, rx=180, rz=-90, shoulder=lefty, elbow=epositive, wrist=wpositive, fatherId=fReference[0]}
  [267] = {x=211, y=-78.226, z=22, rx=180, rz=-90, shoulder=lefty, elbow=epositive, wrist=wpositive, fatherId=fReference[0]}
  [268] = {x=211, y=-88.28, z=22, rx=180, rz=-90, shoulder=lefty, elbow=epositive, wrist=wpositive, fatherId=fReference[0]}
  [269] = {x=211, y=-98.333, z=22, rx=180, rz=-90, shoulder=lefty, elbow=epositive, wrist=wpositive, fatherId=fReference[0]}
  [270] = {x=211, y=-108.386, z=22, rx=180, rz=-90, shoulder=lefty, elbow=epositive, wrist=wpositive, fatherId=fReference[0]}
  [271] = {x=211, y=-118.44, z=22, rx=180, rz=-90, shoulder=lefty, elbow=epositive, wrist=wpositive, fatherId=fReference[0]}
  [272] = {x=211, y=-128.493, z=22, rx=180, rz=-90, shoulder=lefty, elbow=epositive, wrist=wpositive, fatherId=fReference[0]}
  [273] = {x=211, y=-138.546, z=22, rx=180, rz=-90, shoulder=lefty, elbow=epositive, wrist=wpositive, fatherId=fReference[0]}
  [274] = {x=211, y=-148.6, z=22, rx=180, rz=-88.43, shoulder=lefty, elbow=epositive, wrist=wpositive, fatherId=fReference[0]}
  [275] = {x=210.725, y=-158.644, z=22, rx=180, rz=-79.45, shoulder=lefty, elbow=epositive, wrist=wpositive, fatherId=fReference[0]}
  [276] = {x=208.886, y=-168.515, z=22, rx=180, rz=-69.519, shoulder=lefty, elbow=epositive, wrist=wpositive, fatherId=fReference[0]}
  [277] = {x=205.373, y=-177.921, z=22, rx=180, rz=-59.588, shoulder=lefty, elbow=epositive, wrist=wpositive, fatherId=fReference[0]}
  [278] = {x=200.29, y=-186.58, z=22, rx=180, rz=-49.656, shoulder=lefty, elbow=epositive, wrist=wpositive, fatherId=fReference[0]}
  [279] = {x=193.79, y=-194.233, z=22, rx=-180, rz=-39.725, shoulder=lefty, elbow=epositive, wrist=wpositive, fatherId=fReference[0]}
  [280] = {x=186.068, y=-200.65, z=22, rx=180, rz=-29.794, shoulder=lefty, elbow=epositive, wrist=wpositive, fatherId=fReference[0]}
  [281] = {x=177.354, y=-205.639, z=22, rx=-180, rz=-19.863, shoulder=lefty, elbow=epositive, wrist=wpositive, fatherId=fReference[0]}
  [282] = {x=167.911, y=-209.051, z=22, rx=-180, rz=-9.931, shoulder=lefty, elbow=epositive, wrist=wpositive, fatherId=fReference[0]}
  [283] = {x=158.02, y=-210.782, z=22, rx=-180, rz=-1.241, shoulder=lefty, elbow=epositive, wrist=wpositive, fatherId=fReference[0]}
  [284] = {x=147.973, y=-211, z=22, rx=-180, shoulder=lefty, elbow=epositive, wrist=wpositive, fatherId=fReference[0]}
  [285] = {x=137.92, y=-211, z=22, rx=-180, shoulder=lefty, elbow=epositive, wrist=wpositive, fatherId=fReference[0]}
  [286] = {x=127.867, y=-211, z=22, rx=-180, shoulder=lefty, elbow=epositive, wrist=wpositive, fatherId=fReference[0]}
  [287] = {x=117.813, y=-211, z=22, rx=-180, shoulder=lefty, elbow=epositive, wrist=wpositive, fatherId=fReference[0]}
  [288] = {x=107.76, y=-211, z=22, rx=-180, shoulder=lefty, elbow=epositive, wrist=wpositive, fatherId=fReference[0]}
  [289] = {x=97.707, y=-211, z=22, rx=-180, shoulder=lefty, elbow=epositive, wrist=wpositive, fatherId=fReference[0]}
  [290] = {x=87.653, y=-211, z=22, rx=180, shoulder=lefty, elbow=epositive, wrist=wpositive, fatherId=fReference[0]}
  [291] = {x=77.6, y=-211, z=22, rx=-180, shoulder=lefty, elbow=epositive, wrist=wpositive, fatherId=fReference[0]}
  [292] = {x=67.547, y=-211, z=22, rx=180, shoulder=lefty, elbow=epositive, wrist=wpositive, fatherId=fReference[0]}
  [293] = {x=57.493, y=-211, z=22, rx=-180, shoulder=lefty, elbow=epositive, wrist=wpositive, fatherId=fReference[0]}
  [294] = {x=47.44, y=-211, z=22, rx=-180, shoulder=lefty, elbow=epositive, wrist=wpositive, fatherId=fReference[0]}
  [295] = {x=37.387, y=-211, z=22, rx=-180, shoulder=lefty, elbow=epositive, wrist=wpositive, fatherId=fReference[0]}
  [296] = {x=27.333, y=-211, z=22, rx=-180, shoulder=lefty, elbow=epositive, wrist=wpositive, fatherId=fReference[0]}
  [297] = {x=17.28, y=-211, z=22, rx=180, shoulder=lefty, elbow=epositive, wrist=wpositive, fatherId=fReference[0]}
  [298] = {x=7.227, y=-211, z=22, rx=-180, shoulder=lefty, elbow=epositive, wrist=wpositive, fatherId=fReference[0]}
  [299] = {x=-2.826, y=-211, z=22, rx=-180, shoulder=lefty, elbow=epositive, wrist=wpositive, fatherId=fReference[0]}
  [300] = {x=-12.88, y=-211, z=22, rx=-180, shoulder=lefty, elbow=epositive, wrist=wpositive, fatherId=fReference[0]}
  [301] = {x=-22.933, y=-211, z=22, rx=-180, shoulder=lefty, elbow=epositive, wrist=wpositive, fatherId=fReference[0]}
  [302] = {x=-32.986, y=-211, z=22, rx=-180, shoulder=lefty, elbow=epositive, wrist=wpositive, fatherId=fReference[0]}
  [303] = {x=-43.04, y=-211, z=22, rx=180, shoulder=lefty, elbow=epositive, wrist=wpositive, fatherId=fReference[0]}
  [304] = {x=-53.093, y=-211, z=22, rx=180, shoulder=lefty, elbow=epositive, wrist=wpositive, fatherId=fReference[0]}
  [305] = {x=-63.146, y=-211, z=22, rx=180, shoulder=lefty, elbow=epositive, wrist=wpositive, fatherId=fReference[0]}
  [306] = {x=-73.2, y=-211, z=22, rx=180, shoulder=lefty, elbow=epositive, wrist=wpositive, fatherId=fReference[0]}
  [307] = {x=-83.253, y=-211, z=22, rx=-180, shoulder=lefty, elbow=epositive, wrist=wpositive, fatherId=fReference[0]}
  [308] = {x=-93.306, y=-211, z=22, rx=-180, shoulder=lefty, elbow=epositive, wrist=wpositive, fatherId=fReference[0]}
  [309] = {x=-103.36, y=-211, z=22, rx=180, shoulder=lefty, elbow=epositive, wrist=wpositive, fatherId=fReference[0]}
  [310] = {x=-113.413, y=-211, z=22, rx=180, shoulder=lefty, elbow=epositive, wrist=wpositive, fatherId=fReference[0]}
  [311] = {x=-123.466, y=-211, z=22, rx=180, shoulder=lefty, elbow=epositive, wrist=wpositive, fatherId=fReference[0]}
  [312] = {x=-133.52, y=-211, z=22, rx=180, shoulder=lefty, elbow=epositive, wrist=wpositive, fatherId=fReference[0]}
  [313] = {x=-143.573, y=-211, z=22, rx=-180, rz=0.019, shoulder=lefty, elbow=epositive, wrist=wpositive, fatherId=fReference[0]}
  [314] = {x=-153.626, y=-210.997, z=22, rx=180, rz=5.584, shoulder=lefty, elbow=epositive, wrist=wpositive, fatherId=fReference[0]}
  [315] = {x=-163.619, y=-210.02, z=22, rx=-180, rz=15.516, shoulder=lefty, elbow=epositive, wrist=wpositive, fatherId=fReference[0]}
  [316] = {x=-173.294, y=-207.334, z=22, rx=-180, rz=25.447, shoulder=lefty, elbow=epositive, wrist=wpositive, fatherId=fReference[0]}
  [317] = {x=-182.361, y=-203.019, z=22, rx=-180, rz=35.378, shoulder=lefty, elbow=epositive, wrist=wpositive, fatherId=fReference[0]}
  [318] = {x=-190.548, y=-197.206, z=22, rx=180, rz=45.309, shoulder=lefty, elbow=epositive, wrist=wpositive, fatherId=fReference[0]}
  [319] = {x=-197.609, y=-190.068, z=22, rx=-180, rz=55.241, shoulder=lefty, elbow=epositive, wrist=wpositive, fatherId=fReference[0]}
  [320] = {x=-203.334, y=-181.819, z=22, rx=-180, rz=65.172, shoulder=lefty, elbow=epositive, wrist=wpositive, fatherId=fReference[0]}
  [321] = {x=-207.55, y=-172.706, z=22, rx=-180, rz=75.103, shoulder=lefty, elbow=epositive, wrist=wpositive, fatherId=fReference[0]}
  [322] = {x=-210.131, y=-163.003, z=22, rx=-180, rz=85.034, shoulder=lefty, elbow=epositive, wrist=wpositive, fatherId=fReference[0]}
  [323] = {x=-211, y=-153, z=22, rx=-180, rz=85.034, shoulder=lefty, elbow=epositive, wrist=wpositive, fatherId=fReference[0]}
  [324] = {x=-211, y=-153, z=22, rx=-180, rz=85.034, shoulder=lefty, elbow=epositive, wrist=wpositive, fatherId=fReference[0]}
  [325] = {x=-211, y=-153, z=122, rx=-180, rz=85.034, shoulder=lefty, elbow=epositive, wrist=wpositive, fatherId=fReference[0]}
  [326] = {x=-211, y=-153, z=144, rx=-180, rz=85.034, shoulder=lefty, elbow=epositive, wrist=wpositive, fatherId=fReference[0]}
  [327] = {x=-211, y=-153, z=44, rx=-180, rz=85.034, shoulder=lefty, elbow=epositive, wrist=wpositive, fatherId=fReference[0]}
  [328] = {x=-211, y=-153, z=44, rx=-180, rz=85.034, shoulder=lefty, elbow=epositive, wrist=wpositive, fatherId=fReference[0]}
  [329] = {x=-210.131, y=-163.003, z=44, rx=-180, rz=75.103, shoulder=lefty, elbow=epositive, wrist=wpositive, fatherId=fReference[0]}
  [330] = {x=-207.55, y=-172.706, z=44, rx=-180, rz=65.172, shoulder=lefty, elbow=epositive, wrist=wpositive, fatherId=fReference[0]}
  [331] = {x=-203.334, y=-181.819, z=44, rx=-180, rz=55.241, shoulder=lefty, elbow=epositive, wrist=wpositive, fatherId=fReference[0]}
  [332] = {x=-197.609, y=-190.068, z=44, rx=-180, rz=45.309, shoulder=lefty, elbow=epositive, wrist=wpositive, fatherId=fReference[0]}
  [333] = {x=-190.548, y=-197.206, z=44, rx=180, rz=35.378, shoulder=lefty, elbow=epositive, wrist=wpositive, fatherId=fReference[0]}
  [334] = {x=-182.361, y=-203.019, z=44, rx=-180, rz=25.447, shoulder=lefty, elbow=epositive, wrist=wpositive, fatherId=fReference[0]}
  [335] = {x=-173.294, y=-207.334, z=44, rx=-180, rz=15.516, shoulder=lefty, elbow=epositive, wrist=wpositive, fatherId=fReference[0]}
  [336] = {x=-163.619, y=-210.02, z=44, rx=-180, rz=5.584, shoulder=lefty, elbow=epositive, wrist=wpositive, fatherId=fReference[0]}
  [337] = {x=-153.626, y=-210.997, z=44, rx=180, rz=0.019, shoulder=lefty, elbow=epositive, wrist=wpositive, fatherId=fReference[0]}
  [338] = {x=-143.573, y=-211, z=44, rx=-180, shoulder=lefty, elbow=epositive, wrist=wpositive, fatherId=fReference[0]}
  [339] = {x=-133.52, y=-211, z=44, rx=180, shoulder=lefty, elbow=epositive, wrist=wpositive, fatherId=fReference[0]}
  [340] = {x=-123.466, y=-211, z=44, rx=-180, shoulder=lefty, elbow=epositive, wrist=wpositive, fatherId=fReference[0]}
  [341] = {x=-113.413, y=-211, z=44, rx=-180, shoulder=lefty, elbow=epositive, wrist=wpositive, fatherId=fReference[0]}
  [342] = {x=-103.36, y=-211, z=44, rx=-180, shoulder=lefty, elbow=epositive, wrist=wpositive, fatherId=fReference[0]}
  [343] = {x=-93.306, y=-211, z=44, rx=180, shoulder=lefty, elbow=epositive, wrist=wpositive, fatherId=fReference[0]}
  [344] = {x=-83.253, y=-211, z=44, rx=-180, shoulder=lefty, elbow=epositive, wrist=wpositive, fatherId=fReference[0]}
  [345] = {x=-73.2, y=-211, z=44, rx=-180, shoulder=lefty, elbow=epositive, wrist=wpositive, fatherId=fReference[0]}
  [346] = {x=-63.146, y=-211, z=44, rx=-180, shoulder=lefty, elbow=epositive, wrist=wpositive, fatherId=fReference[0]}
  [347] = {x=-53.093, y=-211, z=44, rx=-180, shoulder=lefty, elbow=epositive, wrist=wpositive, fatherId=fReference[0]}
  [348] = {x=-43.04, y=-211, z=44, rx=180, shoulder=lefty, elbow=epositive, wrist=wpositive, fatherId=fReference[0]}
  [349] = {x=-32.986, y=-211, z=44, rx=-180, shoulder=lefty, elbow=epositive, wrist=wpositive, fatherId=fReference[0]}
  [350] = {x=-22.933, y=-211, z=44, rx=-180, shoulder=lefty, elbow=epositive, wrist=wpositive, fatherId=fReference[0]}
  [351] = {x=-12.88, y=-211, z=44, rx=180, shoulder=lefty, elbow=epositive, wrist=wpositive, fatherId=fReference[0]}
  [352] = {x=-2.826, y=-211, z=44, rx=180, shoulder=lefty, elbow=epositive, wrist=wpositive, fatherId=fReference[0]}
  [353] = {x=7.227, y=-211, z=44, rx=180, shoulder=lefty, elbow=epositive, wrist=wpositive, fatherId=fReference[0]}
  [354] = {x=17.28, y=-211, z=44, rx=180, shoulder=lefty, elbow=epositive, wrist=wpositive, fatherId=fReference[0]}
  [355] = {x=27.333, y=-211, z=44, rx=-180, shoulder=lefty, elbow=epositive, wrist=wpositive, fatherId=fReference[0]}
  [356] = {x=37.387, y=-211, z=44, rx=-180, shoulder=lefty, elbow=epositive, wrist=wpositive, fatherId=fReference[0]}
  [357] = {x=47.44, y=-211, z=44, rx=180, shoulder=lefty, elbow=epositive, wrist=wpositive, fatherId=fReference[0]}
  [358] = {x=57.493, y=-211, z=44, rx=-180, shoulder=lefty, elbow=epositive, wrist=wpositive, fatherId=fReference[0]}
  [359] = {x=67.547, y=-211, z=44, rx=180, shoulder=lefty, elbow=epositive, wrist=wpositive, fatherId=fReference[0]}
  [360] = {x=77.6, y=-211, z=44, rx=-180, shoulder=lefty, elbow=epositive, wrist=wpositive, fatherId=fReference[0]}
  [361] = {x=87.653, y=-211, z=44, rx=-180, shoulder=lefty, elbow=epositive, wrist=wpositive, fatherId=fReference[0]}
  [362] = {x=97.707, y=-211, z=44, rx=-180, shoulder=lefty, elbow=epositive, wrist=wpositive, fatherId=fReference[0]}
  [363] = {x=107.76, y=-211, z=44, rx=-180, shoulder=lefty, elbow=epositive, wrist=wpositive, fatherId=fReference[0]}
  [364] = {x=117.813, y=-211, z=44, rx=-180, shoulder=lefty, elbow=epositive, wrist=wpositive, fatherId=fReference[0]}
  [365] = {x=127.867, y=-211, z=44, rx=-180, shoulder=lefty, elbow=epositive, wrist=wpositive, fatherId=fReference[0]}
  [366] = {x=137.92, y=-211, z=44, rx=-180, shoulder=lefty, elbow=epositive, wrist=wpositive, fatherId=fReference[0]}
  [367] = {x=147.973, y=-211, z=44, rx=-180, rz=-1.241, shoulder=lefty, elbow=epositive, wrist=wpositive, fatherId=fReference[0]}
  [368] = {x=158.02, y=-210.782, z=44, rx=180, rz=-9.931, shoulder=lefty, elbow=epositive, wrist=wpositive, fatherId=fReference[0]}
  [369] = {x=167.911, y=-209.051, z=44, rx=180, rz=-19.863, shoulder=lefty, elbow=epositive, wrist=wpositive, fatherId=fReference[0]}
  [370] = {x=177.354, y=-205.639, z=44, rx=-180, rz=-29.794, shoulder=lefty, elbow=epositive, wrist=wpositive, fatherId=fReference[0]}
  [371] = {x=186.068, y=-200.65, z=44, rx=-180, rz=-39.725, shoulder=lefty, elbow=epositive, wrist=wpositive, fatherId=fReference[0]}
  [372] = {x=193.79, y=-194.233, z=44, rx=180, rz=-49.656, shoulder=lefty, elbow=epositive, wrist=wpositive, fatherId=fReference[0]}
  [373] = {x=200.29, y=-186.58, z=44, rx=180, rz=-59.588, shoulder=lefty, elbow=epositive, wrist=wpositive, fatherId=fReference[0]}
  [374] = {x=205.373, y=-177.921, z=44, rx=180, rz=-69.519, shoulder=lefty, elbow=epositive, wrist=wpositive, fatherId=fReference[0]}
  [375] = {x=208.886, y=-168.515, z=44, rx=180, rz=-79.45, shoulder=lefty, elbow=epositive, wrist=wpositive, fatherId=fReference[0]}
  [376] = {x=210.725, y=-158.644, z=44, rx=180, rz=-88.43, shoulder=lefty, elbow=epositive, wrist=wpositive, fatherId=fReference[0]}
  [377] = {x=211, y=-148.6, z=44, rx=180, rz=-90, shoulder=lefty, elbow=epositive, wrist=wpositive, fatherId=fReference[0]}
  [378] = {x=211, y=-138.546, z=44, rx=180, rz=-90, shoulder=lefty, elbow=epositive, wrist=wpositive, fatherId=fReference[0]}
  [379] = {x=211, y=-128.493, z=44, rx=180, rz=-90, shoulder=lefty, elbow=epositive, wrist=wpositive, fatherId=fReference[0]}
  [380] = {x=211, y=-118.44, z=44, rx=180, rz=-90, shoulder=lefty, elbow=epositive, wrist=wpositive, fatherId=fReference[0]}
  [381] = {x=211, y=-108.386, z=44, rx=180, rz=-90, shoulder=lefty, elbow=epositive, wrist=wpositive, fatherId=fReference[0]}
  [382] = {x=211, y=-98.333, z=44, rx=180, rz=-90, shoulder=lefty, elbow=epositive, wrist=wpositive, fatherId=fReference[0]}
  [383] = {x=211, y=-88.28, z=44, rx=180, rz=-90, shoulder=lefty, elbow=epositive, wrist=wpositive, fatherId=fReference[0]}
  [384] = {x=211, y=-78.226, z=44, rx=180, rz=-90, shoulder=lefty, elbow=epositive, wrist=wpositive, fatherId=fReference[0]}
  [385] = {x=211, y=-68.173, z=44, rx=180, rz=-90, shoulder=lefty, elbow=epositive, wrist=wpositive, fatherId=fReference[0]}
  [386] = {x=211, y=-58.12, z=44, rx=180, rz=-90, shoulder=lefty, elbow=epositive, wrist=wpositive, fatherId=fReference[0]}
  [387] = {x=211, y=-48.066, z=44, rx=180, rz=-90, shoulder=lefty, elbow=epositive, wrist=wpositive, fatherId=fReference[0]}
  [388] = {x=211, y=-38.013, z=44, rx=180, rz=-90, shoulder=lefty, elbow=epositive, wrist=wpositive, fatherId=fReference[0]}
  [389] = {x=211, y=-27.96, z=44, rx=180, rz=-90, shoulder=lefty, elbow=epositive, wrist=wpositive, fatherId=fReference[0]}
  [390] = {x=211, y=-17.906, z=44, rx=180, rz=-90, shoulder=lefty, elbow=epositive, wrist=wpositive, fatherId=fReference[0]}
  [391] = {x=211, y=-7.853, z=44, rx=180, rz=-90, shoulder=lefty, elbow=epositive, wrist=wpositive, fatherId=fReference[0]}
  [392] = {x=211, y=2.2, z=44, rx=180, rz=-90, shoulder=lefty, elbow=epositive, wrist=wpositive, fatherId=fReference[0]}
  [393] = {x=211, y=12.254, z=44, rx=180, rz=-90, shoulder=lefty, elbow=epositive, wrist=wpositive, fatherId=fReference[0]}
  [394] = {x=211, y=22.307, z=44, rx=180, rz=-90, shoulder=lefty, elbow=epositive, wrist=wpositive, fatherId=fReference[0]}
  [395] = {x=211, y=32.36, z=44, rx=180, rz=-90, shoulder=lefty, elbow=epositive, wrist=wpositive, fatherId=fReference[0]}
  [396] = {x=211, y=42.413, z=44, rx=180, rz=-90, shoulder=lefty, elbow=epositive, wrist=wpositive, fatherId=fReference[0]}
  [397] = {x=211, y=52.467, z=44, rx=180, rz=-90, shoulder=lefty, elbow=epositive, wrist=wpositive, fatherId=fReference[0]}
  [398] = {x=211, y=62.52, z=44, rx=180, rz=-90, shoulder=lefty, elbow=epositive, wrist=wpositive, fatherId=fReference[0]}
  [399] = {x=211, y=72.573, z=44, rx=180, rz=-90, shoulder=lefty, elbow=epositive, wrist=wpositive, fatherId=fReference[0]}
  [400] = {x=211, y=82.627, z=44, rx=180, rz=-90, shoulder=lefty, elbow=epositive, wrist=wpositive, fatherId=fReference[0]}
  [401] = {x=211, y=92.68, z=44, rx=180, rz=-90, shoulder=lefty, elbow=epositive, wrist=wpositive, fatherId=fReference[0]}
  [402] = {x=211, y=102.733, z=44, rx=180, rz=-90, shoulder=lefty, elbow=epositive, wrist=wpositive, fatherId=fReference[0]}
  [403] = {x=211, y=112.787, z=44, rx=180, rz=-90, shoulder=lefty, elbow=epositive, wrist=wpositive, fatherId=fReference[0]}
  [404] = {x=211, y=122.84, z=44, rx=180, rz=-90, shoulder=lefty, elbow=epositive, wrist=wpositive, fatherId=fReference[0]}
  [405] = {x=211, y=132.893, z=44, rx=180, rz=-90, shoulder=lefty, elbow=epositive, wrist=wpositive, fatherId=fReference[0]}
  [406] = {x=211, y=142.947, z=44, rx=180, rz=-90, shoulder=lefty, elbow=epositive, wrist=wpositive, fatherId=fReference[0]}
  [407] = {x=211, y=153, z=44, rx=-180, rz=-94.966, shoulder=lefty, elbow=epositive, wrist=wpositive, fatherId=fReference[0]}
  [408] = {x=210.131, y=163.003, z=44, rx=-180, rz=-104.897, shoulder=lefty, elbow=epositive, wrist=wpositive, fatherId=fReference[0]}
  [409] = {x=207.55, y=172.706, z=44, rx=-180, rz=-114.828, shoulder=lefty, elbow=epositive, wrist=wpositive, fatherId=fReference[0]}
  [410] = {x=203.334, y=181.819, z=44, rx=-180, rz=-124.759, shoulder=lefty, elbow=epositive, wrist=wpositive, fatherId=fReference[0]}
  [411] = {x=197.609, y=190.068, z=44, rx=-180, rz=-134.691, shoulder=lefty, elbow=epositive, wrist=wpositive, fatherId=fReference[0]}
  [412] = {x=190.548, y=197.206, z=44, rx=-180, rz=-144.622, shoulder=lefty, elbow=epositive, wrist=wpositive, fatherId=fReference[0]}
  [413] = {x=182.361, y=203.019, z=44, rx=-180, rz=-154.553, shoulder=lefty, elbow=epositive, wrist=wpositive, fatherId=fReference[0]}
  [414] = {x=173.294, y=207.334, z=44, rx=-180, rz=-164.484, shoulder=lefty, elbow=epositive, wrist=wpositive, fatherId=fReference[0]}
  [415] = {x=163.619, y=210.02, z=44, rx=-180, rz=-174.416, shoulder=lefty, elbow=epositive, wrist=wpositive, fatherId=fReference[0]}
  [416] = {x=153.626, y=210.997, z=44, rx=180, rz=-179.981, shoulder=lefty, elbow=epositive, wrist=wpositive, fatherId=fReference[0]}
  [417] = {x=143.573, y=211, z=44, rx=-180, rz=-180, shoulder=lefty, elbow=epositive, wrist=wpositive, fatherId=fReference[0]}
  [418] = {x=133.52, y=211, z=44, rx=-180, rz=-180, shoulder=lefty, elbow=epositive, wrist=wpositive, fatherId=fReference[0]}
  [419] = {x=123.466, y=211, z=44, rx=-180, rz=-180, shoulder=lefty, elbow=epositive, wrist=wpositive, fatherId=fReference[0]}
  [420] = {x=113.413, y=211, z=44, rx=180, rz=-180, shoulder=lefty, elbow=epositive, wrist=wpositive, fatherId=fReference[0]}
  [421] = {x=103.36, y=211, z=44, rx=-180, rz=-180, shoulder=lefty, elbow=epositive, wrist=wpositive, fatherId=fReference[0]}
  [422] = {x=93.306, y=211, z=44, rx=180, rz=-180, shoulder=lefty, elbow=epositive, wrist=wpositive, fatherId=fReference[0]}
  [423] = {x=83.253, y=211, z=44, rx=180, rz=-180, shoulder=lefty, elbow=epositive, wrist=wpositive, fatherId=fReference[0]}
  [424] = {x=73.2, y=211, z=44, rx=-180, rz=-180, shoulder=lefty, elbow=epositive, wrist=wpositive, fatherId=fReference[0]}
  [425] = {x=63.146, y=211, z=44, rx=180, rz=-180, shoulder=lefty, elbow=epositive, wrist=wpositive, fatherId=fReference[0]}
  [426] = {x=53.093, y=211, z=44, rx=180, rz=-180, shoulder=lefty, elbow=epositive, wrist=wpositive, fatherId=fReference[0]}
  [427] = {x=43.04, y=211, z=44, rx=180, rz=-180, shoulder=lefty, elbow=epositive, wrist=wpositive, fatherId=fReference[0]}
  [428] = {x=32.986, y=211, z=44, rx=-180, rz=-180, shoulder=lefty, elbow=epositive, wrist=wpositive, fatherId=fReference[0]}
  [429] = {x=22.933, y=211, z=44, rx=180, rz=-180, shoulder=lefty, elbow=epositive, wrist=wpositive, fatherId=fReference[0]}
  [430] = {x=12.88, y=211, z=44, rx=180, rz=-180, shoulder=lefty, elbow=epositive, wrist=wpositive, fatherId=fReference[0]}
  [431] = {x=2.826, y=211, z=44, rx=180, rz=-180, shoulder=lefty, elbow=epositive, wrist=wpositive, fatherId=fReference[0]}
  [432] = {x=-7.227, y=211, z=44, rx=-180, rz=-180, shoulder=lefty, elbow=epositive, wrist=wpositive, fatherId=fReference[0]}
  [433] = {x=-17.28, y=211, z=44, rx=-180, rz=-180, shoulder=lefty, elbow=epositive, wrist=wpositive, fatherId=fReference[0]}
  [434] = {x=-27.333, y=211, z=44, rx=180, rz=-180, shoulder=lefty, elbow=epositive, wrist=wpositive, fatherId=fReference[0]}
  [435] = {x=-37.387, y=211, z=44, rx=-180, rz=-180, shoulder=lefty, elbow=epositive, wrist=wpositive, fatherId=fReference[0]}
  [436] = {x=-47.44, y=211, z=44, rx=180, rz=-180, shoulder=lefty, elbow=epositive, wrist=wpositive, fatherId=fReference[0]}
  [437] = {x=-57.493, y=211, z=44, rx=-180, rz=-180, shoulder=lefty, elbow=epositive, wrist=wpositive, fatherId=fReference[0]}
  [438] = {x=-67.547, y=211, z=44, rx=180, rz=-180, shoulder=lefty, elbow=epositive, wrist=wpositive, fatherId=fReference[0]}
  [439] = {x=-77.6, y=211, z=44, rx=-180, rz=-180, shoulder=lefty, elbow=epositive, wrist=wpositive, fatherId=fReference[0]}
  [440] = {x=-87.653, y=211, z=44, rx=-180, rz=-180, shoulder=lefty, elbow=epositive, wrist=wpositive, fatherId=fReference[0]}
  [441] = {x=-97.707, y=211, z=44, rx=180, rz=-180, shoulder=lefty, elbow=epositive, wrist=wpositive, fatherId=fReference[0]}
  [442] = {x=-107.76, y=211, z=44, rx=-180, rz=-180, shoulder=lefty, elbow=epositive, wrist=wpositive, fatherId=fReference[0]}
  [443] = {x=-117.813, y=211, z=44, rx=180, rz=-180, shoulder=lefty, elbow=epositive, wrist=wpositive, fatherId=fReference[0]}
  [444] = {x=-127.867, y=211, z=44, rx=-180, rz=-180, shoulder=lefty, elbow=epositive, wrist=wpositive, fatherId=fReference[0]}
  [445] = {x=-137.92, y=211, z=44, rx=180, rz=-180, shoulder=lefty, elbow=epositive, wrist=wpositive, fatherId=fReference[0]}
  [446] = {x=-147.973, y=211, z=44, rx=180, rz=178.759, shoulder=lefty, elbow=epositive, wrist=wpositive, fatherId=fReference[0]}
  [447] = {x=-158.02, y=210.782, z=44, rx=180, rz=170.069, shoulder=lefty, elbow=epositive, wrist=wpositive, fatherId=fReference[0]}
  [448] = {x=-167.911, y=209.051, z=44, rx=180, rz=160.137, shoulder=lefty, elbow=epositive, wrist=wpositive, fatherId=fReference[0]}
  [449] = {x=-177.354, y=205.639, z=44, rx=180, rz=150.206, shoulder=lefty, elbow=epositive, wrist=wpositive, fatherId=fReference[0]}
  [450] = {x=-186.068, y=200.65, z=44, rx=180, rz=140.275, shoulder=lefty, elbow=epositive, wrist=wpositive, fatherId=fReference[0]}
  [451] = {x=-193.79, y=194.233, z=44, rx=180, rz=130.344, shoulder=lefty, elbow=epositive, wrist=wpositive, fatherId=fReference[0]}
  [452] = {x=-200.29, y=186.58, z=44, rx=180, rz=120.412, shoulder=lefty, elbow=epositive, wrist=wpositive, fatherId=fReference[0]}
  [453] = {x=-205.373, y=177.921, z=44, rx=180, rz=110.481, shoulder=lefty, elbow=epositive, wrist=wpositive, fatherId=fReference[0]}
  [454] = {x=-208.886, y=168.515, z=44, rx=180, rz=100.55, shoulder=lefty, elbow=epositive, wrist=wpositive, fatherId=fReference[0]}
  [455] = {x=-210.725, y=158.644, z=44, rx=180, rz=91.57, shoulder=lefty, elbow=epositive, wrist=wpositive, fatherId=fReference[0]}
  [456] = {x=-211, y=148.6, z=44, rx=180, rz=90, shoulder=lefty, elbow=epositive, wrist=wpositive, fatherId=fReference[0]}
  [457] = {x=-211, y=138.546, z=44, rx=180, rz=90, shoulder=lefty, elbow=epositive, wrist=wpositive, fatherId=fReference[0]}
  [458] = {x=-211, y=128.493, z=44, rx=180, rz=90, shoulder=lefty, elbow=epositive, wrist=wpositive, fatherId=fReference[0]}
  [459] = {x=-211, y=118.44, z=44, rx=180, rz=90, shoulder=lefty, elbow=epositive, wrist=wpositive, fatherId=fReference[0]}
  [460] = {x=-211, y=108.386, z=44, rx=180, rz=90, shoulder=lefty, elbow=epositive, wrist=wpositive, fatherId=fReference[0]}
  [461] = {x=-211, y=98.333, z=44, rx=180, rz=90, shoulder=lefty, elbow=epositive, wrist=wpositive, fatherId=fReference[0]}
  [462] = {x=-211, y=88.28, z=44, rx=180, rz=90, shoulder=lefty, elbow=epositive, wrist=wpositive, fatherId=fReference[0]}
  [463] = {x=-211, y=78.226, z=44, rx=180, rz=90, shoulder=lefty, elbow=epositive, wrist=wpositive, fatherId=fReference[0]}
  [464] = {x=-211, y=68.173, z=44, rx=180, rz=90, shoulder=lefty, elbow=epositive, wrist=wpositive, fatherId=fReference[0]}
  [465] = {x=-211, y=58.12, z=44, rx=180, rz=90, shoulder=lefty, elbow=epositive, wrist=wpositive, fatherId=fReference[0]}
  [466] = {x=-211, y=48.066, z=44, rx=180, rz=90, shoulder=lefty, elbow=epositive, wrist=wpositive, fatherId=fReference[0]}
  [467] = {x=-211, y=38.013, z=44, rx=180, rz=90, shoulder=lefty, elbow=epositive, wrist=wpositive, fatherId=fReference[0]}
  [468] = {x=-211, y=27.96, z=44, rx=180, rz=90, shoulder=lefty, elbow=epositive, wrist=wpositive, fatherId=fReference[0]}
  [469] = {x=-211, y=17.906, z=44, rx=180, rz=90, shoulder=lefty, elbow=epositive, wrist=wpositive, fatherId=fReference[0]}
  [470] = {x=-211, y=7.853, z=44, rx=180, rz=90, shoulder=lefty, elbow=epositive, wrist=wpositive, fatherId=fReference[0]}
  [471] = {x=-211, y=-2.2, z=44, rx=180, rz=90, shoulder=lefty, elbow=epositive, wrist=wpositive, fatherId=fReference[0]}
  [472] = {x=-211, y=-12.254, z=44, rx=180, rz=90, shoulder=lefty, elbow=epositive, wrist=wpositive, fatherId=fReference[0]}
  [473] = {x=-211, y=-22.307, z=44, rx=180, rz=90, shoulder=lefty, elbow=epositive, wrist=wpositive, fatherId=fReference[0]}
  [474] = {x=-211, y=-32.36, z=44, rx=180, rz=90, shoulder=lefty, elbow=epositive, wrist=wpositive, fatherId=fReference[0]}
  [475] = {x=-211, y=-42.413, z=44, rx=180, rz=90, shoulder=lefty, elbow=epositive, wrist=wpositive, fatherId=fReference[0]}
  [476] = {x=-211, y=-52.467, z=44, rx=180, rz=90, shoulder=lefty, elbow=epositive, wrist=wpositive, fatherId=fReference[0]}
  [477] = {x=-211, y=-62.52, z=44, rx=180, rz=90, shoulder=lefty, elbow=epositive, wrist=wpositive, fatherId=fReference[0]}
  [478] = {x=-211, y=-72.573, z=44, rx=180, rz=90, shoulder=lefty, elbow=epositive, wrist=wpositive, fatherId=fReference[0]}
  [479] = {x=-211, y=-82.627, z=44, rx=180, rz=90, shoulder=lefty, elbow=epositive, wrist=wpositive, fatherId=fReference[0]}
  [480] = {x=-211, y=-92.68, z=44, rx=180, rz=90, shoulder=lefty, elbow=epositive, wrist=wpositive, fatherId=fReference[0]}
  [481] = {x=-211, y=-102.733, z=44, rx=180, rz=90, shoulder=lefty, elbow=epositive, wrist=wpositive, fatherId=fReference[0]}
  [482] = {x=-211, y=-112.787, z=44, rx=180, rz=90, shoulder=lefty, elbow=epositive, wrist=wpositive, fatherId=fReference[0]}
  [483] = {x=-211, y=-122.84, z=44, rx=180, rz=90, shoulder=lefty, elbow=epositive, wrist=wpositive, fatherId=fReference[0]}
  [484] = {x=-211, y=-132.893, z=44, rx=180, rz=90, shoulder=lefty, elbow=epositive, wrist=wpositive, fatherId=fReference[0]}
  [485] = {x=-211, y=-142.947, z=44, rx=180, rz=90, shoulder=lefty, elbow=epositive, wrist=wpositive, fatherId=fReference[0]}
  [486] = {x=-211, y=-153, z=44, rx=180, rz=90, shoulder=lefty, elbow=epositive, wrist=wpositive, fatherId=fReference[0]}
  [487] = {x=-211, y=-153, z=44, rx=180, rz=90, shoulder=lefty, elbow=epositive, wrist=wpositive, fatherId=fReference[0]}
  [488] = {x=-211, y=-153, z=144, rx=180, rz=90, shoulder=lefty, elbow=epositive, wrist=wpositive, fatherId=fReference[0]}
  [489] = {x=-211, y=-153, z=166, rx=180, rz=90, shoulder=lefty, elbow=epositive, wrist=wpositive, fatherId=fReference[0]}
  [490] = {x=-211, y=-153, z=66, rx=180, rz=90, shoulder=lefty, elbow=epositive, wrist=wpositive, fatherId=fReference[0]}
  [491] = {x=-211, y=-153, z=66, rx=180, rz=90, shoulder=lefty, elbow=epositive, wrist=wpositive, fatherId=fReference[0]}
  [492] = {x=-211, y=-142.947, z=66, rx=180, rz=90, shoulder=lefty, elbow=epositive, wrist=wpositive, fatherId=fReference[0]}
  [493] = {x=-211, y=-132.893, z=66, rx=180, rz=90, shoulder=lefty, elbow=epositive, wrist=wpositive, fatherId=fReference[0]}
  [494] = {x=-211, y=-122.84, z=66, rx=180, rz=90, shoulder=lefty, elbow=epositive, wrist=wpositive, fatherId=fReference[0]}
  [495] = {x=-211, y=-112.787, z=66, rx=180, rz=90, shoulder=lefty, elbow=epositive, wrist=wpositive, fatherId=fReference[0]}
  [496] = {x=-211, y=-102.733, z=66, rx=180, rz=90, shoulder=lefty, elbow=epositive, wrist=wpositive, fatherId=fReference[0]}
  [497] = {x=-211, y=-92.68, z=66, rx=180, rz=90, shoulder=lefty, elbow=epositive, wrist=wpositive, fatherId=fReference[0]}
  [498] = {x=-211, y=-82.627, z=66, rx=180, rz=90, shoulder=lefty, elbow=epositive, wrist=wpositive, fatherId=fReference[0]}
  [499] = {x=-211, y=-72.573, z=66, rx=180, rz=90, shoulder=lefty, elbow=epositive, wrist=wpositive, fatherId=fReference[0]}
  [500] = {x=-211, y=-62.52, z=66, rx=180, rz=90, shoulder=lefty, elbow=epositive, wrist=wpositive, fatherId=fReference[0]}
  [501] = {x=-211, y=-52.467, z=66, rx=180, rz=90, shoulder=lefty, elbow=epositive, wrist=wpositive, fatherId=fReference[0]}
  [502] = {x=-211, y=-42.413, z=66, rx=180, rz=90, shoulder=lefty, elbow=epositive, wrist=wpositive, fatherId=fReference[0]}
  [503] = {x=-211, y=-32.36, z=66, rx=180, rz=90, shoulder=lefty, elbow=epositive, wrist=wpositive, fatherId=fReference[0]}
  [504] = {x=-211, y=-22.307, z=66, rx=180, rz=90, shoulder=lefty, elbow=epositive, wrist=wpositive, fatherId=fReference[0]}
  [505] = {x=-211, y=-12.254, z=66, rx=180, rz=90, shoulder=lefty, elbow=epositive, wrist=wpositive, fatherId=fReference[0]}
  [506] = {x=-211, y=-2.2, z=66, rx=180, rz=90, shoulder=lefty, elbow=epositive, wrist=wpositive, fatherId=fReference[0]}
  [507] = {x=-211, y=7.853, z=66, rx=180, rz=90, shoulder=lefty, elbow=epositive, wrist=wpositive, fatherId=fReference[0]}
  [508] = {x=-211, y=17.906, z=66, rx=180, rz=90, shoulder=lefty, elbow=epositive, wrist=wpositive, fatherId=fReference[0]}
  [509] = {x=-211, y=27.96, z=66, rx=180, rz=90, shoulder=lefty, elbow=epositive, wrist=wpositive, fatherId=fReference[0]}
  [510] = {x=-211, y=38.013, z=66, rx=180, rz=90, shoulder=lefty, elbow=epositive, wrist=wpositive, fatherId=fReference[0]}
  [511] = {x=-211, y=48.066, z=66, rx=180, rz=90, shoulder=lefty, elbow=epositive, wrist=wpositive, fatherId=fReference[0]}
  [512] = {x=-211, y=58.12, z=66, rx=180, rz=90, shoulder=lefty, elbow=epositive, wrist=wpositive, fatherId=fReference[0]}
  [513] = {x=-211, y=68.173, z=66, rx=180, rz=90, shoulder=lefty, elbow=epositive, wrist=wpositive, fatherId=fReference[0]}
  [514] = {x=-211, y=78.226, z=66, rx=180, rz=90, shoulder=lefty, elbow=epositive, wrist=wpositive, fatherId=fReference[0]}
  [515] = {x=-211, y=88.28, z=66, rx=180, rz=90, shoulder=lefty, elbow=epositive, wrist=wpositive, fatherId=fReference[0]}
  [516] = {x=-211, y=98.333, z=66, rx=180, rz=90, shoulder=lefty, elbow=epositive, wrist=wpositive, fatherId=fReference[0]}
  [517] = {x=-211, y=108.386, z=66, rx=180, rz=90, shoulder=lefty, elbow=epositive, wrist=wpositive, fatherId=fReference[0]}
  [518] = {x=-211, y=118.44, z=66, rx=180, rz=90, shoulder=lefty, elbow=epositive, wrist=wpositive, fatherId=fReference[0]}
  [519] = {x=-211, y=128.493, z=66, rx=180, rz=90, shoulder=lefty, elbow=epositive, wrist=wpositive, fatherId=fReference[0]}
  [520] = {x=-211, y=138.546, z=66, rx=180, rz=90, shoulder=lefty, elbow=epositive, wrist=wpositive, fatherId=fReference[0]}
  [521] = {x=-211, y=148.6, z=66, rx=180, rz=91.57, shoulder=lefty, elbow=epositive, wrist=wpositive, fatherId=fReference[0]}
  [522] = {x=-210.725, y=158.644, z=66, rx=180, rz=100.55, shoulder=lefty, elbow=epositive, wrist=wpositive, fatherId=fReference[0]}
  [523] = {x=-208.886, y=168.515, z=66, rx=180, rz=110.481, shoulder=lefty, elbow=epositive, wrist=wpositive, fatherId=fReference[0]}
  [524] = {x=-205.373, y=177.921, z=66, rx=180, rz=120.412, shoulder=lefty, elbow=epositive, wrist=wpositive, fatherId=fReference[0]}
  [525] = {x=-200.29, y=186.58, z=66, rx=180, rz=130.344, shoulder=lefty, elbow=epositive, wrist=wpositive, fatherId=fReference[0]}
  [526] = {x=-193.79, y=194.233, z=66, rx=180, rz=140.275, shoulder=lefty, elbow=epositive, wrist=wpositive, fatherId=fReference[0]}
  [527] = {x=-186.068, y=200.65, z=66, rx=180, rz=150.206, shoulder=lefty, elbow=epositive, wrist=wpositive, fatherId=fReference[0]}
  [528] = {x=-177.354, y=205.639, z=66, rx=180, rz=160.137, shoulder=lefty, elbow=epositive, wrist=wpositive, fatherId=fReference[0]}
  [529] = {x=-167.911, y=209.051, z=66, rx=-180, rz=170.069, shoulder=lefty, elbow=epositive, wrist=wpositive, fatherId=fReference[0]}
  [530] = {x=-158.02, y=210.782, z=66, rx=-180, rz=178.759, shoulder=lefty, elbow=epositive, wrist=wpositive, fatherId=fReference[0]}
  [531] = {x=-147.973, y=211, z=66, rx=-180, rz=-180, shoulder=lefty, elbow=epositive, wrist=wpositive, fatherId=fReference[0]}
  [532] = {x=-137.92, y=211, z=66, rx=-180, rz=-180, shoulder=lefty, elbow=epositive, wrist=wpositive, fatherId=fReference[0]}
  [533] = {x=-127.867, y=211, z=66, rx=180, rz=-180, shoulder=lefty, elbow=epositive, wrist=wpositive, fatherId=fReference[0]}
  [534] = {x=-117.813, y=211, z=66, rx=-180, rz=-180, shoulder=lefty, elbow=epositive, wrist=wpositive, fatherId=fReference[0]}
  [535] = {x=-107.76, y=211, z=66, rx=180, rz=-180, shoulder=lefty, elbow=epositive, wrist=wpositive, fatherId=fReference[0]}
  [536] = {x=-97.707, y=211, z=66, rx=180, rz=-180, shoulder=lefty, elbow=epositive, wrist=wpositive, fatherId=fReference[0]}
  [537] = {x=-87.653, y=211, z=66, rx=-180, rz=-180, shoulder=lefty, elbow=epositive, wrist=wpositive, fatherId=fReference[0]}
  [538] = {x=-77.6, y=211, z=66, rx=-180, rz=-180, shoulder=lefty, elbow=epositive, wrist=wpositive, fatherId=fReference[0]}
  [539] = {x=-67.547, y=211, z=66, rx=180, rz=-180, shoulder=lefty, elbow=epositive, wrist=wpositive, fatherId=fReference[0]}
  [540] = {x=-57.493, y=211, z=66, rx=180, rz=-180, shoulder=lefty, elbow=epositive, wrist=wpositive, fatherId=fReference[0]}
  [541] = {x=-47.44, y=211, z=66, rx=-180, rz=-180, shoulder=lefty, elbow=epositive, wrist=wpositive, fatherId=fReference[0]}
  [542] = {x=-37.387, y=211, z=66, rx=-180, rz=-180, shoulder=lefty, elbow=epositive, wrist=wpositive, fatherId=fReference[0]}
  [543] = {x=-27.333, y=211, z=66, rx=180, rz=-180, shoulder=lefty, elbow=epositive, wrist=wpositive, fatherId=fReference[0]}
  [544] = {x=-17.28, y=211, z=66, rx=-180, rz=-180, shoulder=lefty, elbow=epositive, wrist=wpositive, fatherId=fReference[0]}
  [545] = {x=-7.227, y=211, z=66, rx=-180, rz=-180, shoulder=lefty, elbow=epositive, wrist=wpositive, fatherId=fReference[0]}
  [546] = {x=2.826, y=211, z=66, rx=-180, rz=-180, shoulder=lefty, elbow=epositive, wrist=wpositive, fatherId=fReference[0]}
  [547] = {x=12.88, y=211, z=66, rx=180, rz=-180, shoulder=lefty, elbow=epositive, wrist=wpositive, fatherId=fReference[0]}
  [548] = {x=22.933, y=211, z=66, rx=180, rz=-180, shoulder=lefty, elbow=epositive, wrist=wpositive, fatherId=fReference[0]}
  [549] = {x=32.986, y=211, z=66, rx=180, rz=-180, shoulder=lefty, elbow=epositive, wrist=wpositive, fatherId=fReference[0]}
  [550] = {x=43.04, y=211, z=66, rx=-180, rz=-180, shoulder=lefty, elbow=epositive, wrist=wpositive, fatherId=fReference[0]}
  [551] = {x=53.093, y=211, z=66, rx=180, rz=-180, shoulder=lefty, elbow=epositive, wrist=wpositive, fatherId=fReference[0]}
  [552] = {x=63.146, y=211, z=66, rx=-180, rz=-180, shoulder=lefty, elbow=epositive, wrist=wpositive, fatherId=fReference[0]}
  [553] = {x=73.2, y=211, z=66, rx=180, rz=-180, shoulder=lefty, elbow=epositive, wrist=wpositive, fatherId=fReference[0]}
  [554] = {x=83.253, y=211, z=66, rx=180, rz=-180, shoulder=lefty, elbow=epositive, wrist=wpositive, fatherId=fReference[0]}
  [555] = {x=93.306, y=211, z=66, rx=-180, rz=-180, shoulder=lefty, elbow=epositive, wrist=wpositive, fatherId=fReference[0]}
  [556] = {x=103.36, y=211, z=66, rx=-180, rz=-180, shoulder=lefty, elbow=epositive, wrist=wpositive, fatherId=fReference[0]}
  [557] = {x=113.413, y=211, z=66, rx=180, rz=-180, shoulder=lefty, elbow=epositive, wrist=wpositive, fatherId=fReference[0]}
  [558] = {x=123.466, y=211, z=66, rx=-180, rz=-180, shoulder=lefty, elbow=epositive, wrist=wpositive, fatherId=fReference[0]}
  [559] = {x=133.52, y=211, z=66, rx=-180, rz=-180, shoulder=lefty, elbow=epositive, wrist=wpositive, fatherId=fReference[0]}
  [560] = {x=143.573, y=211, z=66, rx=-180, rz=-179.981, shoulder=lefty, elbow=epositive, wrist=wpositive, fatherId=fReference[0]}
  [561] = {x=153.626, y=210.997, z=66, rx=-180, rz=-174.416, shoulder=lefty, elbow=epositive, wrist=wpositive, fatherId=fReference[0]}
  [562] = {x=163.619, y=210.02, z=66, rx=180, rz=-164.484, shoulder=lefty, elbow=epositive, wrist=wpositive, fatherId=fReference[0]}
  [563] = {x=173.294, y=207.334, z=66, rx=180, rz=-154.553, shoulder=lefty, elbow=epositive, wrist=wpositive, fatherId=fReference[0]}
  [564] = {x=182.361, y=203.019, z=66, rx=-180, rz=-144.622, shoulder=lefty, elbow=epositive, wrist=wpositive, fatherId=fReference[0]}
  [565] = {x=190.548, y=197.206, z=66, rx=-180, rz=-134.691, shoulder=lefty, elbow=epositive, wrist=wpositive, fatherId=fReference[0]}
  [566] = {x=197.609, y=190.068, z=66, rx=-180, rz=-124.759, shoulder=lefty, elbow=epositive, wrist=wpositive, fatherId=fReference[0]}
  [567] = {x=203.334, y=181.819, z=66, rx=-180, rz=-114.828, shoulder=lefty, elbow=epositive, wrist=wpositive, fatherId=fReference[0]}
  [568] = {x=207.55, y=172.706, z=66, rx=-180, rz=-104.897, shoulder=lefty, elbow=epositive, wrist=wpositive, fatherId=fReference[0]}
  [569] = {x=210.131, y=163.003, z=66, rx=-180, rz=-94.966, shoulder=lefty, elbow=epositive, wrist=wpositive, fatherId=fReference[0]}
  [570] = {x=211, y=153, z=66, rx=180, rz=-90, shoulder=lefty, elbow=epositive, wrist=wpositive, fatherId=fReference[0]}
  [571] = {x=211, y=142.947, z=66, rx=180, rz=-90, shoulder=lefty, elbow=epositive, wrist=wpositive, fatherId=fReference[0]}
  [572] = {x=211, y=132.893, z=66, rx=180, rz=-90, shoulder=lefty, elbow=epositive, wrist=wpositive, fatherId=fReference[0]}
  [573] = {x=211, y=122.84, z=66, rx=180, rz=-90, shoulder=lefty, elbow=epositive, wrist=wpositive, fatherId=fReference[0]}
  [574] = {x=211, y=112.787, z=66, rx=180, rz=-90, shoulder=lefty, elbow=epositive, wrist=wpositive, fatherId=fReference[0]}
  [575] = {x=211, y=102.733, z=66, rx=180, rz=-90, shoulder=lefty, elbow=epositive, wrist=wpositive, fatherId=fReference[0]}
  [576] = {x=211, y=92.68, z=66, rx=180, rz=-90, shoulder=lefty, elbow=epositive, wrist=wpositive, fatherId=fReference[0]}
  [577] = {x=211, y=82.627, z=66, rx=180, rz=-90, shoulder=lefty, elbow=epositive, wrist=wpositive, fatherId=fReference[0]}
  [578] = {x=211, y=72.573, z=66, rx=180, rz=-90, shoulder=lefty, elbow=epositive, wrist=wpositive, fatherId=fReference[0]}
  [579] = {x=211, y=62.52, z=66, rx=180, rz=-90, shoulder=lefty, elbow=epositive, wrist=wpositive, fatherId=fReference[0]}
  [580] = {x=211, y=52.467, z=66, rx=180, rz=-90, shoulder=lefty, elbow=epositive, wrist=wpositive, fatherId=fReference[0]}
  [581] = {x=211, y=42.413, z=66, rx=180, rz=-90, shoulder=lefty, elbow=epositive, wrist=wpositive, fatherId=fReference[0]}
  [582] = {x=211, y=32.36, z=66, rx=180, rz=-90, shoulder=lefty, elbow=epositive, wrist=wpositive, fatherId=fReference[0]}
  [583] = {x=211, y=22.307, z=66, rx=180, rz=-90, shoulder=lefty, elbow=epositive, wrist=wpositive, fatherId=fReference[0]}
  [584] = {x=211, y=12.254, z=66, rx=180, rz=-90, shoulder=lefty, elbow=epositive, wrist=wpositive, fatherId=fReference[0]}
  [585] = {x=211, y=2.2, z=66, rx=180, rz=-90, shoulder=lefty, elbow=epositive, wrist=wpositive, fatherId=fReference[0]}
  [586] = {x=211, y=-7.853, z=66, rx=180, rz=-90, shoulder=lefty, elbow=epositive, wrist=wpositive, fatherId=fReference[0]}
  [587] = {x=211, y=-17.906, z=66, rx=180, rz=-90, shoulder=lefty, elbow=epositive, wrist=wpositive, fatherId=fReference[0]}
  [588] = {x=211, y=-27.96, z=66, rx=180, rz=-90, shoulder=lefty, elbow=epositive, wrist=wpositive, fatherId=fReference[0]}
  [589] = {x=211, y=-38.013, z=66, rx=180, rz=-90, shoulder=lefty, elbow=epositive, wrist=wpositive, fatherId=fReference[0]}
  [590] = {x=211, y=-48.066, z=66, rx=180, rz=-90, shoulder=lefty, elbow=epositive, wrist=wpositive, fatherId=fReference[0]}
  [591] = {x=211, y=-58.12, z=66, rx=180, rz=-90, shoulder=lefty, elbow=epositive, wrist=wpositive, fatherId=fReference[0]}
  [592] = {x=211, y=-68.173, z=66, rx=180, rz=-90, shoulder=lefty, elbow=epositive, wrist=wpositive, fatherId=fReference[0]}
  [593] = {x=211, y=-78.226, z=66, rx=180, rz=-90, shoulder=lefty, elbow=epositive, wrist=wpositive, fatherId=fReference[0]}
  [594] = {x=211, y=-88.28, z=66, rx=180, rz=-90, shoulder=lefty, elbow=epositive, wrist=wpositive, fatherId=fReference[0]}
  [595] = {x=211, y=-98.333, z=66, rx=180, rz=-90, shoulder=lefty, elbow=epositive, wrist=wpositive, fatherId=fReference[0]}
  [596] = {x=211, y=-108.386, z=66, rx=180, rz=-90, shoulder=lefty, elbow=epositive, wrist=wpositive, fatherId=fReference[0]}
  [597] = {x=211, y=-118.44, z=66, rx=180, rz=-90, shoulder=lefty, elbow=epositive, wrist=wpositive, fatherId=fReference[0]}
  [598] = {x=211, y=-128.493, z=66, rx=180, rz=-90, shoulder=lefty, elbow=epositive, wrist=wpositive, fatherId=fReference[0]}
  [599] = {x=211, y=-138.546, z=66, rx=180, rz=-90, shoulder=lefty, elbow=epositive, wrist=wpositive, fatherId=fReference[0]}
  [600] = {x=211, y=-148.6, z=66, rx=180, rz=-88.43, shoulder=lefty, elbow=epositive, wrist=wpositive, fatherId=fReference[0]}
  [601] = {x=210.725, y=-158.644, z=66, rx=-180, rz=-79.45, shoulder=lefty, elbow=epositive, wrist=wpositive, fatherId=fReference[0]}
  [602] = {x=208.886, y=-168.515, z=66, rx=180, rz=-69.519, shoulder=lefty, elbow=epositive, wrist=wpositive, fatherId=fReference[0]}
  [603] = {x=205.373, y=-177.921, z=66, rx=180, rz=-59.588, shoulder=lefty, elbow=epositive, wrist=wpositive, fatherId=fReference[0]}
  [604] = {x=200.29, y=-186.58, z=66, rx=180, rz=-49.656, shoulder=lefty, elbow=epositive, wrist=wpositive, fatherId=fReference[0]}
  [605] = {x=193.79, y=-194.233, z=66, rx=180, rz=-39.725, shoulder=lefty, elbow=epositive, wrist=wpositive, fatherId=fReference[0]}
  [606] = {x=186.068, y=-200.65, z=66, rx=-180, rz=-29.794, shoulder=lefty, elbow=epositive, wrist=wpositive, fatherId=fReference[0]}
  [607] = {x=177.354, y=-205.639, z=66, rx=180, rz=-19.863, shoulder=lefty, elbow=epositive, wrist=wpositive, fatherId=fReference[0]}
  [608] = {x=167.911, y=-209.051, z=66, rx=-180, rz=-9.931, shoulder=lefty, elbow=epositive, wrist=wpositive, fatherId=fReference[0]}
  [609] = {x=158.02, y=-210.782, z=66, rx=-180, rz=-1.241, shoulder=lefty, elbow=epositive, wrist=wpositive, fatherId=fReference[0]}
  [610] = {x=147.973, y=-211, z=66, rx=180, shoulder=lefty, elbow=epositive, wrist=wpositive, fatherId=fReference[0]}
  [611] = {x=137.92, y=-211, z=66, rx=-180, shoulder=lefty, elbow=epositive, wrist=wpositive, fatherId=fReference[0]}
  [612] = {x=127.867, y=-211, z=66, rx=-180, shoulder=lefty, elbow=epositive, wrist=wpositive, fatherId=fReference[0]}
  [613] = {x=117.813, y=-211, z=66, rx=-180, shoulder=lefty, elbow=epositive, wrist=wpositive, fatherId=fReference[0]}
  [614] = {x=107.76, y=-211, z=66, rx=-180, shoulder=lefty, elbow=epositive, wrist=wpositive, fatherId=fReference[0]}
  [615] = {x=97.707, y=-211, z=66, rx=-180, shoulder=lefty, elbow=epositive, wrist=wpositive, fatherId=fReference[0]}
  [616] = {x=87.653, y=-211, z=66, rx=-180, shoulder=lefty, elbow=epositive, wrist=wpositive, fatherId=fReference[0]}
  [617] = {x=77.6, y=-211, z=66, rx=-180, shoulder=lefty, elbow=epositive, wrist=wpositive, fatherId=fReference[0]}
  [618] = {x=67.547, y=-211, z=66, rx=180, shoulder=lefty, elbow=epositive, wrist=wpositive, fatherId=fReference[0]}
  [619] = {x=57.493, y=-211, z=66, rx=-180, shoulder=lefty, elbow=epositive, wrist=wpositive, fatherId=fReference[0]}
  [620] = {x=47.44, y=-211, z=66, rx=180, shoulder=lefty, elbow=epositive, wrist=wpositive, fatherId=fReference[0]}
  [621] = {x=37.387, y=-211, z=66, rx=180, shoulder=lefty, elbow=epositive, wrist=wpositive, fatherId=fReference[0]}
  [622] = {x=27.333, y=-211, z=66, rx=-180, shoulder=lefty, elbow=epositive, wrist=wpositive, fatherId=fReference[0]}
  [623] = {x=17.28, y=-211, z=66, rx=180, shoulder=lefty, elbow=epositive, wrist=wpositive, fatherId=fReference[0]}
  [624] = {x=7.227, y=-211, z=66, rx=180, shoulder=lefty, elbow=epositive, wrist=wpositive, fatherId=fReference[0]}
  [625] = {x=-2.826, y=-211, z=66, rx=-180, shoulder=lefty, elbow=epositive, wrist=wpositive, fatherId=fReference[0]}
  [626] = {x=-12.88, y=-211, z=66, rx=-180, shoulder=lefty, elbow=epositive, wrist=wpositive, fatherId=fReference[0]}
  [627] = {x=-22.933, y=-211, z=66, rx=-180, shoulder=lefty, elbow=epositive, wrist=wpositive, fatherId=fReference[0]}
  [628] = {x=-32.986, y=-211, z=66, rx=-180, shoulder=lefty, elbow=epositive, wrist=wpositive, fatherId=fReference[0]}
  [629] = {x=-43.04, y=-211, z=66, rx=-180, shoulder=lefty, elbow=epositive, wrist=wpositive, fatherId=fReference[0]}
  [630] = {x=-53.093, y=-211, z=66, rx=180, shoulder=lefty, elbow=epositive, wrist=wpositive, fatherId=fReference[0]}
  [631] = {x=-63.146, y=-211, z=66, rx=-180, shoulder=lefty, elbow=epositive, wrist=wpositive, fatherId=fReference[0]}
  [632] = {x=-73.2, y=-211, z=66, rx=-180, shoulder=lefty, elbow=epositive, wrist=wpositive, fatherId=fReference[0]}
  [633] = {x=-83.253, y=-211, z=66, rx=180, shoulder=lefty, elbow=epositive, wrist=wpositive, fatherId=fReference[0]}
  [634] = {x=-93.306, y=-211, z=66, rx=-180, shoulder=lefty, elbow=epositive, wrist=wpositive, fatherId=fReference[0]}
  [635] = {x=-103.36, y=-211, z=66, rx=-180, shoulder=lefty, elbow=epositive, wrist=wpositive, fatherId=fReference[0]}
  [636] = {x=-113.413, y=-211, z=66, rx=180, shoulder=lefty, elbow=epositive, wrist=wpositive, fatherId=fReference[0]}
  [637] = {x=-123.466, y=-211, z=66, rx=-180, shoulder=lefty, elbow=epositive, wrist=wpositive, fatherId=fReference[0]}
  [638] = {x=-133.52, y=-211, z=66, rx=-180, shoulder=lefty, elbow=epositive, wrist=wpositive, fatherId=fReference[0]}
  [639] = {x=-143.573, y=-211, z=66, rx=180, rz=0.019, shoulder=lefty, elbow=epositive, wrist=wpositive, fatherId=fReference[0]}
  [640] = {x=-153.626, y=-210.997, z=66, rx=-180, rz=5.584, shoulder=lefty, elbow=epositive, wrist=wpositive, fatherId=fReference[0]}
  [641] = {x=-163.619, y=-210.02, z=66, rx=-180, rz=15.516, shoulder=lefty, elbow=epositive, wrist=wpositive, fatherId=fReference[0]}
  [642] = {x=-173.294, y=-207.334, z=66, rx=-180, rz=25.447, shoulder=lefty, elbow=epositive, wrist=wpositive, fatherId=fReference[0]}
  [643] = {x=-182.361, y=-203.019, z=66, rx=-180, rz=35.378, shoulder=lefty, elbow=epositive, wrist=wpositive, fatherId=fReference[0]}
  [644] = {x=-190.548, y=-197.206, z=66, rx=-180, rz=45.309, shoulder=lefty, elbow=epositive, wrist=wpositive, fatherId=fReference[0]}
  [645] = {x=-197.609, y=-190.068, z=66, rx=180, rz=55.241, shoulder=lefty, elbow=epositive, wrist=wpositive, fatherId=fReference[0]}
  [646] = {x=-203.334, y=-181.819, z=66, rx=-180, rz=65.172, shoulder=lefty, elbow=epositive, wrist=wpositive, fatherId=fReference[0]}
  [647] = {x=-207.55, y=-172.706, z=66, rx=-180, rz=75.103, shoulder=lefty, elbow=epositive, wrist=wpositive, fatherId=fReference[0]}
  [648] = {x=-210.131, y=-163.003, z=66, rx=-180, rz=85.034, shoulder=lefty, elbow=epositive, wrist=wpositive, fatherId=fReference[0]}
  [649] = {x=-211, y=-153, z=66, rx=-180, rz=85.034, shoulder=lefty, elbow=epositive, wrist=wpositive, fatherId=fReference[0]}
  [650] = {x=-211, y=-153, z=66, rx=-180, rz=85.034, shoulder=lefty, elbow=epositive, wrist=wpositive, fatherId=fReference[0]}
  [651] = {x=-211, y=-153, z=166, rx=-180, rz=85.034, shoulder=lefty, elbow=epositive, wrist=wpositive, fatherId=fReference[0]}
  [652] = {x=-211, y=-153, z=188, rx=-180, rz=85.034, shoulder=lefty, elbow=epositive, wrist=wpositive, fatherId=fReference[0]}
  [653] = {x=-211, y=-153, z=88, rx=-180, rz=85.034, shoulder=lefty, elbow=epositive, wrist=wpositive, fatherId=fReference[0]}
  [654] = {x=-211, y=-153, z=88, rx=-180, rz=85.034, shoulder=lefty, elbow=epositive, wrist=wpositive, fatherId=fReference[0]}
  [655] = {x=-210.131, y=-163.003, z=88, rx=-180, rz=75.103, shoulder=lefty, elbow=epositive, wrist=wpositive, fatherId=fReference[0]}
  [656] = {x=-207.55, y=-172.706, z=88, rx=-180, rz=65.172, shoulder=lefty, elbow=epositive, wrist=wpositive, fatherId=fReference[0]}
  [657] = {x=-203.334, y=-181.819, z=88, rx=-180, rz=55.241, shoulder=lefty, elbow=epositive, wrist=wpositive, fatherId=fReference[0]}
  [658] = {x=-197.609, y=-190.068, z=88, rx=180, rz=45.309, shoulder=lefty, elbow=epositive, wrist=wpositive, fatherId=fReference[0]}
  [659] = {x=-190.548, y=-197.206, z=88, rx=-180, rz=35.378, shoulder=lefty, elbow=epositive, wrist=wpositive, fatherId=fReference[0]}
  [660] = {x=-182.361, y=-203.019, z=88, rx=180, rz=25.447, shoulder=lefty, elbow=epositive, wrist=wpositive, fatherId=fReference[0]}
  [661] = {x=-173.294, y=-207.334, z=88, rx=180, rz=15.516, shoulder=lefty, elbow=epositive, wrist=wpositive, fatherId=fReference[0]}
  [662] = {x=-163.619, y=-210.02, z=88, rx=-180, rz=5.584, shoulder=lefty, elbow=epositive, wrist=wpositive, fatherId=fReference[0]}
  [663] = {x=-153.626, y=-210.997, z=88, rx=180, rz=0.019, shoulder=lefty, elbow=epositive, wrist=wpositive, fatherId=fReference[0]}
  [664] = {x=-143.573, y=-211, z=88, rx=180, shoulder=lefty, elbow=epositive, wrist=wpositive, fatherId=fReference[0]}
  [665] = {x=-133.52, y=-211, z=88, rx=180, shoulder=lefty, elbow=epositive, wrist=wpositive, fatherId=fReference[0]}
  [666] = {x=-123.466, y=-211, z=88, rx=-180, shoulder=lefty, elbow=epositive, wrist=wpositive, fatherId=fReference[0]}
  [667] = {x=-113.413, y=-211, z=88, rx=-180, shoulder=lefty, elbow=epositive, wrist=wpositive, fatherId=fReference[0]}
  [668] = {x=-103.36, y=-211, z=88, rx=-180, shoulder=lefty, elbow=epositive, wrist=wpositive, fatherId=fReference[0]}
  [669] = {x=-93.306, y=-211, z=88, rx=-180, shoulder=lefty, elbow=epositive, wrist=wpositive, fatherId=fReference[0]}
  [670] = {x=-83.253, y=-211, z=88, rx=180, shoulder=lefty, elbow=epositive, wrist=wpositive, fatherId=fReference[0]}
  [671] = {x=-73.2, y=-211, z=88, rx=-180, shoulder=lefty, elbow=epositive, wrist=wpositive, fatherId=fReference[0]}
  [672] = {x=-63.146, y=-211, z=88, rx=180, shoulder=lefty, elbow=epositive, wrist=wpositive, fatherId=fReference[0]}
  [673] = {x=-53.093, y=-211, z=88, rx=180, shoulder=lefty, elbow=epositive, wrist=wpositive, fatherId=fReference[0]}
  [674] = {x=-43.04, y=-211, z=88, rx=-180, shoulder=lefty, elbow=epositive, wrist=wpositive, fatherId=fReference[0]}
  [675] = {x=-32.986, y=-211, z=88, rx=-180, shoulder=lefty, elbow=epositive, wrist=wpositive, fatherId=fReference[0]}
  [676] = {x=-22.933, y=-211, z=88, rx=180, shoulder=lefty, elbow=epositive, wrist=wpositive, fatherId=fReference[0]}
  [677] = {x=-12.88, y=-211, z=88, rx=-180, shoulder=lefty, elbow=epositive, wrist=wpositive, fatherId=fReference[0]}
  [678] = {x=-2.826, y=-211, z=88, rx=180, shoulder=lefty, elbow=epositive, wrist=wpositive, fatherId=fReference[0]}
  [679] = {x=7.227, y=-211, z=88, rx=-180, shoulder=lefty, elbow=epositive, wrist=wpositive, fatherId=fReference[0]}
  [680] = {x=17.28, y=-211, z=88, rx=-180, shoulder=lefty, elbow=epositive, wrist=wpositive, fatherId=fReference[0]}
  [681] = {x=27.333, y=-211, z=88, rx=180, shoulder=lefty, elbow=epositive, wrist=wpositive, fatherId=fReference[0]}
  [682] = {x=37.387, y=-211, z=88, rx=-180, shoulder=lefty, elbow=epositive, wrist=wpositive, fatherId=fReference[0]}
  [683] = {x=47.44, y=-211, z=88, rx=180, shoulder=lefty, elbow=epositive, wrist=wpositive, fatherId=fReference[0]}
  [684] = {x=57.493, y=-211, z=88, rx=180, shoulder=lefty, elbow=epositive, wrist=wpositive, fatherId=fReference[0]}
  [685] = {x=67.547, y=-211, z=88, rx=-180, shoulder=lefty, elbow=epositive, wrist=wpositive, fatherId=fReference[0]}
  [686] = {x=77.6, y=-211, z=88, rx=180, shoulder=lefty, elbow=epositive, wrist=wpositive, fatherId=fReference[0]}
  [687] = {x=87.653, y=-211, z=88, rx=180, shoulder=lefty, elbow=epositive, wrist=wpositive, fatherId=fReference[0]}
  [688] = {x=97.707, y=-211, z=88, rx=-180, shoulder=lefty, elbow=epositive, wrist=wpositive, fatherId=fReference[0]}
  [689] = {x=107.76, y=-211, z=88, rx=180, shoulder=lefty, elbow=epositive, wrist=wpositive, fatherId=fReference[0]}
  [690] = {x=117.813, y=-211, z=88, rx=180, shoulder=lefty, elbow=epositive, wrist=wpositive, fatherId=fReference[0]}
  [691] = {x=127.867, y=-211, z=88, rx=180, shoulder=lefty, elbow=epositive, wrist=wpositive, fatherId=fReference[0]}
  [692] = {x=137.92, y=-211, z=88, rx=-180, shoulder=lefty, elbow=epositive, wrist=wpositive, fatherId=fReference[0]}
  [693] = {x=147.973, y=-211, z=88, rx=-180, rz=-1.241, shoulder=lefty, elbow=epositive, wrist=wpositive, fatherId=fReference[0]}
  [694] = {x=158.02, y=-210.782, z=88, rx=-180, rz=-9.931, shoulder=lefty, elbow=epositive, wrist=wpositive, fatherId=fReference[0]}
  [695] = {x=167.911, y=-209.051, z=88, rx=180, rz=-19.863, shoulder=lefty, elbow=epositive, wrist=wpositive, fatherId=fReference[0]}
  [696] = {x=177.354, y=-205.639, z=88, rx=180, rz=-29.794, shoulder=lefty, elbow=epositive, wrist=wpositive, fatherId=fReference[0]}
  [697] = {x=186.068, y=-200.65, z=88, rx=180, rz=-39.725, shoulder=lefty, elbow=epositive, wrist=wpositive, fatherId=fReference[0]}
  [698] = {x=193.79, y=-194.233, z=88, rx=-180, rz=-49.656, shoulder=lefty, elbow=epositive, wrist=wpositive, fatherId=fReference[0]}
  [699] = {x=200.29, y=-186.58, z=88, rx=180, rz=-59.588, shoulder=lefty, elbow=epositive, wrist=wpositive, fatherId=fReference[0]}
  [700] = {x=205.373, y=-177.921, z=88, rx=180, rz=-69.519, shoulder=lefty, elbow=epositive, wrist=wpositive, fatherId=fReference[0]}
  [701] = {x=208.886, y=-168.515, z=88, rx=180, rz=-79.45, shoulder=lefty, elbow=epositive, wrist=wpositive, fatherId=fReference[0]}
  [702] = {x=210.725, y=-158.644, z=88, rx=180, rz=-88.43, shoulder=lefty, elbow=epositive, wrist=wpositive, fatherId=fReference[0]}
  [703] = {x=211, y=-148.6, z=88, rx=180, rz=-90, shoulder=lefty, elbow=epositive, wrist=wpositive, fatherId=fReference[0]}
  [704] = {x=211, y=-138.546, z=88, rx=180, rz=-90, shoulder=lefty, elbow=epositive, wrist=wpositive, fatherId=fReference[0]}
  [705] = {x=211, y=-128.493, z=88, rx=180, rz=-90, shoulder=lefty, elbow=epositive, wrist=wpositive, fatherId=fReference[0]}
  [706] = {x=211, y=-118.44, z=88, rx=180, rz=-90, shoulder=lefty, elbow=epositive, wrist=wpositive, fatherId=fReference[0]}
  [707] = {x=211, y=-108.386, z=88, rx=180, rz=-90, shoulder=lefty, elbow=epositive, wrist=wpositive, fatherId=fReference[0]}
  [708] = {x=211, y=-98.333, z=88, rx=180, rz=-90, shoulder=lefty, elbow=epositive, wrist=wpositive, fatherId=fReference[0]}
  [709] = {x=211, y=-88.28, z=88, rx=180, rz=-90, shoulder=lefty, elbow=epositive, wrist=wpositive, fatherId=fReference[0]}
  [710] = {x=211, y=-78.226, z=88, rx=180, rz=-90, shoulder=lefty, elbow=epositive, wrist=wpositive, fatherId=fReference[0]}
  [711] = {x=211, y=-68.173, z=88, rx=180, rz=-90, shoulder=lefty, elbow=epositive, wrist=wpositive, fatherId=fReference[0]}
  [712] = {x=211, y=-58.12, z=88, rx=180, rz=-90, shoulder=lefty, elbow=epositive, wrist=wpositive, fatherId=fReference[0]}
  [713] = {x=211, y=-48.066, z=88, rx=180, rz=-90, shoulder=lefty, elbow=epositive, wrist=wpositive, fatherId=fReference[0]}
  [714] = {x=211, y=-38.013, z=88, rx=180, rz=-90, shoulder=lefty, elbow=epositive, wrist=wpositive, fatherId=fReference[0]}
  [715] = {x=211, y=-27.96, z=88, rx=180, rz=-90, shoulder=lefty, elbow=epositive, wrist=wpositive, fatherId=fReference[0]}
  [716] = {x=211, y=-17.906, z=88, rx=180, rz=-90, shoulder=lefty, elbow=epositive, wrist=wpositive, fatherId=fReference[0]}
  [717] = {x=211, y=-7.853, z=88, rx=180, rz=-90, shoulder=lefty, elbow=epositive, wrist=wpositive, fatherId=fReference[0]}
  [718] = {x=211, y=2.2, z=88, rx=180, rz=-90, shoulder=lefty, elbow=epositive, wrist=wpositive, fatherId=fReference[0]}
  [719] = {x=211, y=12.254, z=88, rx=180, rz=-90, shoulder=lefty, elbow=epositive, wrist=wpositive, fatherId=fReference[0]}
  [720] = {x=211, y=22.307, z=88, rx=180, rz=-90, shoulder=lefty, elbow=epositive, wrist=wpositive, fatherId=fReference[0]}
  [721] = {x=211, y=32.36, z=88, rx=180, rz=-90, shoulder=lefty, elbow=epositive, wrist=wpositive, fatherId=fReference[0]}
  [722] = {x=211, y=42.413, z=88, rx=180, rz=-90, shoulder=lefty, elbow=epositive, wrist=wpositive, fatherId=fReference[0]}
  [723] = {x=211, y=52.467, z=88, rx=180, rz=-90, shoulder=lefty, elbow=epositive, wrist=wpositive, fatherId=fReference[0]}
  [724] = {x=211, y=62.52, z=88, rx=180, rz=-90, shoulder=lefty, elbow=epositive, wrist=wpositive, fatherId=fReference[0]}
  [725] = {x=211, y=72.573, z=88, rx=180, rz=-90, shoulder=lefty, elbow=epositive, wrist=wpositive, fatherId=fReference[0]}
  [726] = {x=211, y=82.627, z=88, rx=180, rz=-90, shoulder=lefty, elbow=epositive, wrist=wpositive, fatherId=fReference[0]}
  [727] = {x=211, y=92.68, z=88, rx=180, rz=-90, shoulder=lefty, elbow=epositive, wrist=wpositive, fatherId=fReference[0]}
  [728] = {x=211, y=102.733, z=88, rx=180, rz=-90, shoulder=lefty, elbow=epositive, wrist=wpositive, fatherId=fReference[0]}
  [729] = {x=211, y=112.787, z=88, rx=180, rz=-90, shoulder=lefty, elbow=epositive, wrist=wpositive, fatherId=fReference[0]}
  [730] = {x=211, y=122.84, z=88, rx=180, rz=-90, shoulder=lefty, elbow=epositive, wrist=wpositive, fatherId=fReference[0]}
  [731] = {x=211, y=132.893, z=88, rx=180, rz=-90, shoulder=lefty, elbow=epositive, wrist=wpositive, fatherId=fReference[0]}
  [732] = {x=211, y=142.947, z=88, rx=180, rz=-90, shoulder=lefty, elbow=epositive, wrist=wpositive, fatherId=fReference[0]}
  [733] = {x=211, y=153, z=88, rx=-180, rz=-94.966, shoulder=lefty, elbow=epositive, wrist=wpositive, fatherId=fReference[0]}
  [734] = {x=210.131, y=163.003, z=88, rx=-180, rz=-104.897, shoulder=lefty, elbow=epositive, wrist=wpositive, fatherId=fReference[0]}
  [735] = {x=207.55, y=172.706, z=88, rx=-180, rz=-114.828, shoulder=lefty, elbow=epositive, wrist=wpositive, fatherId=fReference[0]}
  [736] = {x=203.334, y=181.819, z=88, rx=-180, rz=-124.759, shoulder=lefty, elbow=epositive, wrist=wpositive, fatherId=fReference[0]}
  [737] = {x=197.609, y=190.068, z=88, rx=-180, rz=-134.691, shoulder=lefty, elbow=epositive, wrist=wpositive, fatherId=fReference[0]}
  [738] = {x=190.548, y=197.206, z=88, rx=180, rz=-144.622, shoulder=lefty, elbow=epositive, wrist=wpositive, fatherId=fReference[0]}
  [739] = {x=182.361, y=203.019, z=88, rx=-180, rz=-154.553, shoulder=lefty, elbow=epositive, wrist=wpositive, fatherId=fReference[0]}
  [740] = {x=173.294, y=207.334, z=88, rx=-180, rz=-164.484, shoulder=lefty, elbow=epositive, wrist=wpositive, fatherId=fReference[0]}
  [741] = {x=163.619, y=210.02, z=88, rx=180, rz=-174.416, shoulder=lefty, elbow=epositive, wrist=wpositive, fatherId=fReference[0]}
  [742] = {x=153.626, y=210.997, z=88, rx=-180, rz=-179.981, shoulder=lefty, elbow=epositive, wrist=wpositive, fatherId=fReference[0]}
  [743] = {x=143.573, y=211, z=88, rx=-180, rz=-180, shoulder=lefty, elbow=epositive, wrist=wpositive, fatherId=fReference[0]}
  [744] = {x=133.52, y=211, z=88, rx=-180, rz=-180, shoulder=lefty, elbow=epositive, wrist=wpositive, fatherId=fReference[0]}
  [745] = {x=123.466, y=211, z=88, rx=180, rz=-180, shoulder=lefty, elbow=epositive, wrist=wpositive, fatherId=fReference[0]}
  [746] = {x=113.413, y=211, z=88, rx=-180, rz=-180, shoulder=lefty, elbow=epositive, wrist=wpositive, fatherId=fReference[0]}
  [747] = {x=103.36, y=211, z=88, rx=180, rz=-180, shoulder=lefty, elbow=epositive, wrist=wpositive, fatherId=fReference[0]}
  [748] = {x=93.306, y=211, z=88, rx=180, rz=-180, shoulder=lefty, elbow=epositive, wrist=wpositive, fatherId=fReference[0]}
  [749] = {x=83.253, y=211, z=88, rx=180, rz=-180, shoulder=lefty, elbow=epositive, wrist=wpositive, fatherId=fReference[0]}
  [750] = {x=73.2, y=211, z=88, rx=180, rz=-180, shoulder=lefty, elbow=epositive, wrist=wpositive, fatherId=fReference[0]}
  [751] = {x=63.146, y=211, z=88, rx=-180, rz=-180, shoulder=lefty, elbow=epositive, wrist=wpositive, fatherId=fReference[0]}
  [752] = {x=53.093, y=211, z=88, rx=180, rz=-180, shoulder=lefty, elbow=epositive, wrist=wpositive, fatherId=fReference[0]}
  [753] = {x=43.04, y=211, z=88, rx=180, rz=-180, shoulder=lefty, elbow=epositive, wrist=wpositive, fatherId=fReference[0]}
  [754] = {x=32.986, y=211, z=88, rx=180, rz=-180, shoulder=lefty, elbow=epositive, wrist=wpositive, fatherId=fReference[0]}
  [755] = {x=22.933, y=211, z=88, rx=180, rz=-180, shoulder=lefty, elbow=epositive, wrist=wpositive, fatherId=fReference[0]}
  [756] = {x=12.88, y=211, z=88, rx=-180, rz=-180, shoulder=lefty, elbow=epositive, wrist=wpositive, fatherId=fReference[0]}
  [757] = {x=2.826, y=211, z=88, rx=180, rz=-180, shoulder=lefty, elbow=epositive, wrist=wpositive, fatherId=fReference[0]}
  [758] = {x=-7.227, y=211, z=88, rx=180, rz=-180, shoulder=lefty, elbow=epositive, wrist=wpositive, fatherId=fReference[0]}
  [759] = {x=-17.28, y=211, z=88, rx=-180, rz=-180, shoulder=lefty, elbow=epositive, wrist=wpositive, fatherId=fReference[0]}
  [760] = {x=-27.333, y=211, z=88, rx=180, rz=-180, shoulder=lefty, elbow=epositive, wrist=wpositive, fatherId=fReference[0]}
  [761] = {x=-37.387, y=211, z=88, rx=180, rz=-180, shoulder=lefty, elbow=epositive, wrist=wpositive, fatherId=fReference[0]}
  [762] = {x=-47.44, y=211, z=88, rx=180, rz=-180, shoulder=lefty, elbow=epositive, wrist=wpositive, fatherId=fReference[0]}
  [763] = {x=-57.493, y=211, z=88, rx=180, rz=-180, shoulder=lefty, elbow=epositive, wrist=wpositive, fatherId=fReference[0]}
  [764] = {x=-67.547, y=211, z=88, rx=180, rz=-180, shoulder=lefty, elbow=epositive, wrist=wpositive, fatherId=fReference[0]}
  [765] = {x=-77.6, y=211, z=88, rx=-180, rz=-180, shoulder=lefty, elbow=epositive, wrist=wpositive, fatherId=fReference[0]}
  [766] = {x=-87.653, y=211, z=88, rx=180, rz=-180, shoulder=lefty, elbow=epositive, wrist=wpositive, fatherId=fReference[0]}
  [767] = {x=-97.707, y=211, z=88, rx=180, rz=-180, shoulder=lefty, elbow=epositive, wrist=wpositive, fatherId=fReference[0]}
  [768] = {x=-107.76, y=211, z=88, rx=180, rz=-180, shoulder=lefty, elbow=epositive, wrist=wpositive, fatherId=fReference[0]}
  [769] = {x=-117.813, y=211, z=88, rx=180, rz=-180, shoulder=lefty, elbow=epositive, wrist=wpositive, fatherId=fReference[0]}
  [770] = {x=-127.867, y=211, z=88, rx=-180, rz=-180, shoulder=lefty, elbow=epositive, wrist=wpositive, fatherId=fReference[0]}
  [771] = {x=-137.92, y=211, z=88, rx=-180, rz=-180, shoulder=lefty, elbow=epositive, wrist=wpositive, fatherId=fReference[0]}
  [772] = {x=-147.973, y=211, z=88, rx=-180, rz=178.759, shoulder=lefty, elbow=epositive, wrist=wpositive, fatherId=fReference[0]}
  [773] = {x=-158.02, y=210.782, z=88, rx=180, rz=170.069, shoulder=lefty, elbow=epositive, wrist=wpositive, fatherId=fReference[0]}
  [774] = {x=-167.911, y=209.051, z=88, rx=180, rz=160.137, shoulder=lefty, elbow=epositive, wrist=wpositive, fatherId=fReference[0]}
  [775] = {x=-177.354, y=205.639, z=88, rx=180, rz=150.206, shoulder=lefty, elbow=epositive, wrist=wpositive, fatherId=fReference[0]}
  [776] = {x=-186.068, y=200.65, z=88, rx=180, rz=140.275, shoulder=lefty, elbow=epositive, wrist=wpositive, fatherId=fReference[0]}
  [777] = {x=-193.79, y=194.233, z=88, rx=180, rz=130.344, shoulder=lefty, elbow=epositive, wrist=wpositive, fatherId=fReference[0]}
  [778] = {x=-200.29, y=186.58, z=88, rx=180, rz=120.412, shoulder=lefty, elbow=epositive, wrist=wpositive, fatherId=fReference[0]}
  [779] = {x=-205.373, y=177.921, z=88, rx=180, rz=110.481, shoulder=lefty, elbow=epositive, wrist=wpositive, fatherId=fReference[0]}
  [780] = {x=-208.886, y=168.515, z=88, rx=180, rz=100.55, shoulder=lefty, elbow=epositive, wrist=wpositive, fatherId=fReference[0]}
  [781] = {x=-210.725, y=158.644, z=88, rx=180, rz=91.57, shoulder=lefty, elbow=epositive, wrist=wpositive, fatherId=fReference[0]}
  [782] = {x=-211, y=148.6, z=88, rx=180, rz=90, shoulder=lefty, elbow=epositive, wrist=wpositive, fatherId=fReference[0]}
  [783] = {x=-211, y=138.546, z=88, rx=180, rz=90, shoulder=lefty, elbow=epositive, wrist=wpositive, fatherId=fReference[0]}
